//     Drive/Outputs/Out/nCtrl2 <-> Receive PDO 1/Control Word @bit 8
//     Drive/Outputs/Out/nDataOut1 <-> Receive PDO 1/Profile Target Position
//     Enc/Inputs/In/nDataIn1 <-> Transmit PDO 1/Position Actual Value
//     Enc/Inputs/In/nDataIn3 <-> Transmit PDO 1/Touch Probe 1 Positive Value
//     Enc/Inputs/In/nDcInputTime <-> InfoData/DcInputShift
//     Enc/Inputs/In/nState4 @bit 1 <-> WcState/InputToggle
//     Enc/Inputs/In/nState4 <-> WcState/WcState
//     Enc/Inputs/In/nState5 <-> Transmit PDO 1/Touch Probe Status
//     Enc/Inputs/In/nState6 <-> Transmit PDO 1/Touch Probe Status @bit 8
//     Enc/Outputs/Out/nCtrl5 <-> Receive PDO 1/Touch Probe Function
//     Enc/Outputs/Out/nCtrl6 <-> Receive PDO 1/Touch Probe Function @bit 8
//   NC-Task 1 SAF/Axes/Axis180_132 P2M3_SCurlingneedleWhirling <-> Device 3 (EtherCAT)/Box 2 (CU1128)/Term 44 (CU1128-C)/P2M3短卷针旋转[132] (CL3C-EC808AC)
//     Drive/Inputs/In/nDcOutputTime <-> InfoData/DcOutputShift
//     Drive/Inputs/In/nState1 <-> Transmit PDO 1/Status Word
//     Drive/Inputs/In/nState2 <-> Transmit PDO 1/Status Word @bit 8
//     Drive/Inputs/In/nState4 @bit 1 <-> WcState/InputToggle
//     Drive/Inputs/In/nState4 <-> WcState/WcState
//     Drive/Outputs/Out/nCtrl1 <-> Receive PDO 1/Control Word
//     Drive/Outputs/Out/nCtrl2 <-> Receive PDO 1/Control Word @bit 8
//     Drive/Outputs/Out/nDataOut1 <-> Receive PDO 1/Profile Target Position
//     Enc/Inputs/In/nDataIn1 <-> Transmit PDO 1/Position Actual Value
//     Enc/Inputs/In/nDataIn3 <-> Transmit PDO 1/Touch Probe 1 Positive Value
//     Enc/Inputs/In/nDcInputTime <-> InfoData/DcInputShift
//     Enc/Inputs/In/nState4 @bit 1 <-> WcState/InputToggle
//     Enc/Inputs/In/nState4 <-> WcState/WcState
//     Enc/Inputs/In/nState5 <-> Transmit PDO 1/Touch Probe Status
//     Enc/Inputs/In/nState6 <-> Transmit PDO 1/Touch Probe Status @bit 8
//     Enc/Outputs/Out/nCtrl5 <-> Receive PDO 1/Touch Probe Function
//     Enc/Outputs/Out/nCtrl6 <-> Receive PDO 1/Touch Probe Function @bit 8
//   NC-Task 1 SAF/Axes/Axis181_133 P2M3_GluingLine <-> Device 3 (EtherCAT)/Box 2 (CU1128)/Term 44 (CU1128-C)/P2M3侧贴夹平移（ 133）(InoSV660N)
//     Drive/Inputs/In/nDataIn1 <-> Inputs/Following error actual value
//     Drive/Inputs/In/nDcOutputTime <-> InfoData/DcOutputShift
//     Drive/Inputs/In/nState1 <-> Inputs/Statusword
//     Drive/Inputs/In/nState2 <-> Inputs/Statusword @bit 8
//     Drive/Inputs/In/nState4 @bit 1 <-> WcState/InputToggle
//     Drive/Inputs/In/nState4 <-> WcState/WcState
//     Drive/Outputs/Out/nCtrl1 <-> Outputs/Controlword
//     Drive/Outputs/Out/nCtrl2 <-> Outputs/Controlword @bit 8
//     Drive/Outputs/Out/nDataOut1 <-> Outputs/Target position
//     Enc/Inputs/In/nDataIn1 <-> Inputs/Position actual value
//     Enc/Inputs/In/nDataIn3 <-> Inputs/Touch probe pos1 pos value
//     Enc/Inputs/In/nDataIn5 <-> Inputs/Touch probe pos2 pos value
//     Enc/Inputs/In/nDcInputTime <-> InfoData/DcInputShift
//     Enc/Inputs/In/nState4 @bit 1 <-> WcState/InputToggle
//     Enc/Inputs/In/nState4 <-> WcState/WcState
//     Enc/Inputs/In/nState5 <-> Inputs/Touch probe status
//     Enc/Inputs/In/nState6 <-> Inputs/Touch probe status @bit 8
//     Enc/Outputs/Out/nCtrl5 <-> Outputs/Touch probe function
//     Enc/Outputs/Out/nCtrl6 <-> Outputs/Touch probe function @bit 8
//   NC-Task 1 SAF/Axes/Axis182_134 P2M3_GluingWhirling <-> Device 3 (EtherCAT)/Box 2 (CU1128)/Term 44 (CU1128-C)/P2M3侧贴夹旋转[134] (InoSV660N)
//     Drive/Inputs/In/nDataIn1 <-> Inputs/Following error actual value
//     Drive/Inputs/In/nDcOutputTime <-> InfoData/DcOutputShift
//     Drive/Inputs/In/nState1 <-> Inputs/Statusword
//     Drive/Inputs/In/nState2 <-> Inputs/Statusword @bit 8
//     Drive/Inputs/In/nState4 @bit 1 <-> WcState/InputToggle
//     Drive/Inputs/In/nState4 <-> WcState/WcState
//     Drive/Outputs/Out/nCtrl1 <-> Outputs/Controlword
//     Drive/Outputs/Out/nCtrl2 <-> Outputs/Controlword @bit 8
//     Drive/Outputs/Out/nDataOut1 <-> Outputs/Target position
//     Enc/Inputs/In/nDataIn1 <-> Inputs/Position actual value
//     Enc/Inputs/In/nDataIn3 <-> Inputs/Touch probe pos1 pos value
//     Enc/Inputs/In/nDataIn5 <-> Inputs/Touch probe pos2 pos value
//     Enc/Inputs/In/nDcInputTime <-> InfoData/DcInputShift
//     Enc/Inputs/In/nState4 @bit 1 <-> WcState/InputToggle
//     Enc/Inputs/In/nState4 <-> WcState/WcState
//     Enc/Inputs/In/nState5 <-> Inputs/Touch probe status
//     Enc/Inputs/In/nState6 <-> Inputs/Touch probe status @bit 8
//     Enc/Outputs/Out/nCtrl5 <-> Outputs/Touch probe function
//     Enc/Outputs/Out/nCtrl6 <-> Outputs/Touch probe function @bit 8
//   NC-Task 1 SAF/Axes/Axis183_135 P2M3_GluingRetracting <-> Device 3 (EtherCAT)/Box 2 (CU1128)/Term 44 (CU1128-C)/P2M3贴胶头进退[135] (InoSV660N)
//     Drive/Inputs/In/nDataIn1 <-> Inputs/Following error actual value
//     Drive/Inputs/In/nDcOutputTime <-> InfoData/DcOutputShift
//     Drive/Inputs/In/nState1 <-> Inputs/Statusword
//     Drive/Inputs/In/nState2 <-> Inputs/Statusword @bit 8
//     Drive/Inputs/In/nState4 @bit 1 <-> WcState/InputToggle
//     Drive/Inputs/In/nState4 <-> WcState/WcState
//     Drive/Outputs/Out/nCtrl1 <-> Outputs/Controlword
//     Drive/Outputs/Out/nCtrl2 <-> Outputs/Controlword @bit 8
//     Drive/Outputs/Out/nDataOut1 <-> Outputs/Target position
//     Enc/Inputs/In/nDataIn1 <-> Inputs/Position actual value
//     Enc/Inputs/In/nDataIn3 <-> Inputs/Touch probe pos1 pos value
//     Enc/Inputs/In/nDataIn5 <-> Inputs/Touch probe pos2 pos value
//     Enc/Inputs/In/nDcInputTime <-> InfoData/DcInputShift
//     Enc/Inputs/In/nState4 @bit 1 <-> WcState/InputToggle
//     Enc/Inputs/In/nState4 <-> WcState/WcState
//     Enc/Inputs/In/nState5 <-> Inputs/Touch probe status
//     Enc/Inputs/In/nState6 <-> Inputs/Touch probe status @bit 8
//     Enc/Outputs/Out/nCtrl5 <-> Outputs/Touch probe function
//     Enc/Outputs/Out/nCtrl6 <-> Outputs/Touch probe function @bit 8
//   NC-Task 1 SAF/Axes/Axis184_136 P2M3_GluingUpDown <-> Device 3 (EtherCAT)/Box 2 (CU1128)/Term 44 (CU1128-C)/P2M3拉胶升降[136](InoSV660N)
//     Drive/Inputs/In/nDataIn1 <-> Inputs/Following error actual value
//     Drive/Inputs/In/nDcOutputTime <-> InfoData/DcOutputShift
//     Drive/Inputs/In/nState1 <-> Inputs/Statusword
//     Drive/Inputs/In/nState2 <-> Inputs/Statusword @bit 8
//     Drive/Inputs/In/nState4 @bit 1 <-> WcState/InputToggle
//     Drive/Inputs/In/nState4 <-> WcState/WcState
//     Drive/Outputs/Out/nCtrl1 <-> Outputs/Controlword
//     Drive/Outputs/Out/nCtrl2 <-> Outputs/Controlword @bit 8
//     Drive/Outputs/Out/nDataOut1 <-> Outputs/Target position
//     Enc/Inputs/In/nDataIn1 <-> Inputs/Position actual value
//     Enc/Inputs/In/nDataIn3 <-> Inputs/Touch probe pos1 pos value
//     Enc/Inputs/In/nDataIn5 <-> Inputs/Touch probe pos2 pos value
//     Enc/Inputs/In/nDcInputTime <-> InfoData/DcInputShift
//     Enc/Inputs/In/nState4 @bit 1 <-> WcState/InputToggle
//     Enc/Inputs/In/nState4 <-> WcState/WcState
//     Enc/Inputs/In/nState5 <-> Inputs/Touch probe status
//     Enc/Inputs/In/nState6 <-> Inputs/Touch probe status @bit 8
//     Enc/Outputs/Out/nCtrl5 <-> Outputs/Touch probe function
//     Enc/Outputs/Out/nCtrl6 <-> Outputs/Touch probe function @bit 8
//   NC-Task 1 SAF/Axes/Axis187_160 P3M1_ColdpreLine <-> Device 3 (EtherCAT)/P2M1冷压上料夹平移 [160（热压）](InoSV660N)
//     Drive/Inputs/In/nDataIn1 <-> Inputs/Following error actual value
//     Drive/Inputs/In/nDcOutputTime <-> InfoData/DcOutputShift
//     Drive/Inputs/In/nState1 <-> Inputs/Statusword
//     Drive/Inputs/In/nState2 <-> Inputs/Statusword @bit 8
//     Drive/Inputs/In/nState4 @bit 1 <-> WcState/InputToggle
//     Drive/Inputs/In/nState4 <-> WcState/WcState
//     Drive/Outputs/Out/nCtrl1 <-> Outputs/Controlword
//     Drive/Outputs/Out/nCtrl2 <-> Outputs/Controlword @bit 8
//     Drive/Outputs/Out/nDataOut1 <-> Outputs/Target position
//     Enc/Inputs/In/nDataIn1 <-> Inputs/Position actual value
//     Enc/Inputs/In/nDataIn3 <-> Inputs/Touch probe pos1 pos value
//     Enc/Inputs/In/nDataIn5 <-> Inputs/Touch probe pos2 pos value
//     Enc/Inputs/In/nDcInputTime <-> InfoData/DcInputShift
//     Enc/Inputs/In/nState4 @bit 1 <-> WcState/InputToggle
//     Enc/Inputs/In/nState4 <-> WcState/WcState
//     Enc/Inputs/In/nState5 <-> Inputs/Touch probe status
//     Enc/Inputs/In/nState6 <-> Inputs/Touch probe status @bit 8
//     Enc/Outputs/Out/nCtrl5 <-> Outputs/Touch probe function
//     Enc/Outputs/Out/nCtrl6 <-> Outputs/Touch probe function @bit 8
//   NC-Task 1 SAF/Axes/Axis188_161 P3M1_ColdpreRetracting <-> Device 3 (EtherCAT)/Box 2 (CU1128)/Term 44 (CU1128-C)/P2M2冷压上料夹进退[161（热压）] (InoSV660N)
//     Drive/Inputs/In/nDataIn1 <-> Inputs/Following error actual value
//     Drive/Inputs/In/nDcOutputTime <-> InfoData/DcOutputShift
//     Drive/Inputs/In/nState1 <-> Inputs/Statusword
//     Drive/Inputs/In/nState2 <-> Inputs/Statusword @bit 8
//     Drive/Inputs/In/nState4 @bit 1 <-> WcState/InputToggle
//     Drive/Inputs/In/nState4 <-> WcState/WcState
//     Drive/Outputs/Out/nCtrl1 <-> Outputs/Controlword
//     Drive/Outputs/Out/nCtrl2 <-> Outputs/Controlword @bit 8
//     Drive/Outputs/Out/nDataOut1 <-> Outputs/Target position
//     Enc/Inputs/In/nDataIn1 <-> Inputs/Position actual value
//     Enc/Inputs/In/nDataIn3 <-> Inputs/Touch probe pos1 pos value
//     Enc/Inputs/In/nDataIn5 <-> Inputs/Touch probe pos2 pos value
//     Enc/Inputs/In/nDcInputTime <-> InfoData/DcInputShift
//     Enc/Inputs/In/nState4 @bit 1 <-> WcState/InputToggle
//     Enc/Inputs/In/nState4 <-> WcState/WcState
//     Enc/Inputs/In/nState5 <-> Inputs/Touch probe status
//     Enc/Inputs/In/nState6 <-> Inputs/Touch probe status @bit 8
//     Enc/Outputs/Out/nCtrl5 <-> Outputs/Touch probe function
//     Enc/Outputs/Out/nCtrl6 <-> Outputs/Touch probe function @bit 8
//   NC-Task 1 SAF/Axes/Axis189_162 P3M1_ColdpreWhirling <-> Device 3 (EtherCAT)/Box 2 (CU1128)/Term 44 (CU1128-C)/P2M2冷压上料夹旋转[162（热压）] (InoSV660N)
//     Drive/Inputs/In/nDataIn1 <-> Inputs/Following error actual value
//     Drive/Inputs/In/nDcOutputTime <-> InfoData/DcOutputShift
//     Drive/Inputs/In/nState1 <-> Inputs/Statusword
//     Drive/Inputs/In/nState2 <-> Inputs/Statusword @bit 8
//     Drive/Inputs/In/nState4 @bit 1 <-> WcState/InputToggle
//     Drive/Inputs/In/nState4 <-> WcState/WcState
//     Drive/Outputs/Out/nCtrl1 <-> Outputs/Controlword
//     Drive/Outputs/Out/nCtrl2 <-> Outputs/Controlword @bit 8
//     Drive/Outputs/Out/nDataOut1 <-> Outputs/Target position
//     Enc/Inputs/In/nDataIn1 <-> Inputs/Position actual value
//     Enc/Inputs/In/nDataIn3 <-> Inputs/Touch probe pos1 pos value
//     Enc/Inputs/In/nDataIn5 <-> Inputs/Touch probe pos2 pos value
//     Enc/Inputs/In/nDcInputTime <-> InfoData/DcInputShift
//     Enc/Inputs/In/nState4 @bit 1 <-> WcState/InputToggle
//     Enc/Inputs/In/nState4 <-> WcState/WcState
//     Enc/Inputs/In/nState5 <-> Inputs/Touch probe status
//     Enc/Inputs/In/nState6 <-> Inputs/Touch probe status @bit 8
//     Enc/Outputs/Out/nCtrl5 <-> Outputs/Touch probe function
//     Enc/Outputs/Out/nCtrl6 <-> Outputs/Touch probe function @bit 8
//   NC-Task 1 SAF/Axes/Axis190_163 P3M1_ColdpreUpDown <-> Device 3 (EtherCAT)/Box 2 (CU1128)/Term 44 (CU1128-C)/P2M2冷压上料夹升降[163（热压）] (InoSV660N)
//     Drive/Inputs/In/nDataIn1 <-> Inputs/Following error actual value
//     Drive/Inputs/In/nDcOutputTime <-> InfoData/DcOutputShift
//     Drive/Inputs/In/nState1 <-> Inputs/Statusword
//     Drive/Inputs/In/nState2 <-> Inputs/Statusword @bit 8
//     Drive/Inputs/In/nState4 @bit 1 <-> WcState/InputToggle
//     Drive/Inputs/In/nState4 <-> WcState/WcState
//     Drive/Outputs/Out/nCtrl1 <-> Outputs/Controlword
//     Drive/Outputs/Out/nCtrl2 <-> Outputs/Controlword @bit 8
//     Drive/Outputs/Out/nDataOut1 <-> Outputs/Target position
//     Enc/Inputs/In/nDataIn1 <-> Inputs/Position actual value
//     Enc/Inputs/In/nDataIn3 <-> Inputs/Touch probe pos1 pos value
//     Enc/Inputs/In/nDataIn5 <-> Inputs/Touch probe pos2 pos value
//     Enc/Inputs/In/nDcInputTime <-> InfoData/DcInputShift
//     Enc/Inputs/In/nState4 @bit 1 <-> WcState/InputToggle
//     Enc/Inputs/In/nState4 <-> WcState/WcState
//     Enc/Inputs/In/nState5 <-> Inputs/Touch probe status
//     Enc/Inputs/In/nState6 <-> Inputs/Touch probe status @bit 8
//     Enc/Outputs/Out/nCtrl5 <-> Outputs/Touch probe function
//     Enc/Outputs/Out/nCtrl6 <-> Outputs/Touch probe function @bit 8
//   NC-Task 1 SAF/Axes/Axis191_164 P3M1_ColdpreSupPlateLine <-> Device 3 (EtherCAT)/Box 2 (CU1128)/Term 24 (CU1128-B)/冷压托板开合[164] (CL3C-EC503)
//     Drive/Inputs/In/nDcOutputTime <-> InfoData/DcOutputShift
//     Drive/Inputs/In/nState1 <-> Transmit PDO 1/Status Word
//     Drive/Inputs/In/nState2 <-> Transmit PDO 1/Status Word @bit 8
//     Drive/Inputs/In/nState4 @bit 1 <-> WcState/InputToggle
//     Drive/Inputs/In/nState4 <-> WcState/WcState
//     Drive/Outputs/Out/nCtrl1 <-> Receive PDO 1/Control Word
//     Drive/Outputs/Out/nCtrl2 <-> Receive PDO 1/Control Word @bit 8
//     Drive/Outputs/Out/nDataOut1 <-> Receive PDO 1/Profile Target Position
//     Enc/Inputs/In/nDataIn1 <-> Transmit PDO 1/Position Actual Value
//     Enc/Inputs/In/nDataIn3 <-> Transmit PDO 1/Touch Probe 1 Positive Value
//     Enc/Inputs/In/nDcInputTime <-> InfoData/DcInputShift
//     Enc/Inputs/In/nState4 @bit 1 <-> WcState/InputToggle
//     Enc/Inputs/In/nState4 <-> WcState/WcState
//     Enc/Inputs/In/nState5 <-> Transmit PDO 1/Touch Probe Status
//     Enc/Inputs/In/nState6 <-> Transmit PDO 1/Touch Probe Status @bit 8
//     Enc/Outputs/Out/nCtrl5 <-> Receive PDO 1/Touch Probe Function
//     Enc/Outputs/Out/nCtrl6 <-> Receive PDO 1/Touch Probe Function @bit 8
//   NC-Task 1 SAF/Axes/Axis192_165 P3M1_ColdpreActuated <-> Device 3 (EtherCAT)/Box 2 (CU1128)/Term 24 (CU1128-B)/冷压驱动[165](InoSV660N)
//     Drive/Inputs/In/nDataIn1 <-> Inputs/Following error actual value
//     Drive/Inputs/In/nDcOutputTime <-> InfoData/DcOutputShift
//     Drive/Inputs/In/nState1 <-> Inputs/Statusword
//     Drive/Inputs/In/nState2 <-> Inputs/Statusword @bit 8
//     Drive/Inputs/In/nState4 @bit 1 <-> WcState/InputToggle
//     Drive/Inputs/In/nState4 <-> WcState/WcState
//     Drive/Outputs/Out/nCtrl1 <-> Outputs/Controlword
//     Drive/Outputs/Out/nCtrl2 <-> Outputs/Controlword @bit 8
//     Drive/Outputs/Out/nDataOut1 <-> Outputs/Target position
//     Enc/Inputs/In/nDataIn1 <-> Inputs/Position actual value
//     Enc/Inputs/In/nDataIn3 <-> Inputs/Touch probe pos1 pos value
//     Enc/Inputs/In/nDataIn5 <-> Inputs/Touch probe pos2 pos value
//     Enc/Inputs/In/nDcInputTime <-> InfoData/DcInputShift
//     Enc/Inputs/In/nState4 @bit 1 <-> WcState/InputToggle
//     Enc/Inputs/In/nState4 <-> WcState/WcState
//     Enc/Inputs/In/nState5 <-> Inputs/Touch probe status
//     Enc/Inputs/In/nState6 <-> Inputs/Touch probe status @bit 8
//     Enc/Outputs/Out/nCtrl5 <-> Outputs/Touch probe function
//     Enc/Outputs/Out/nCtrl6 <-> Outputs/Touch probe function @bit 8
//   NC-Task 1 SAF/Axes/Axis193_166 P3_M2_OvenCarrying <-> Device 3 (EtherCAT)/Box 2 (CU1128)/Term 24 (CU1128-B)/烤箱上料夹搬运[166] (InoSV660N)
//     Drive/Inputs/In/nDataIn1 <-> Inputs/Following error actual value
//     Drive/Inputs/In/nDcOutputTime <-> InfoData/DcOutputShift
//     Drive/Inputs/In/nState1 <-> Inputs/Statusword
//     Drive/Inputs/In/nState2 <-> Inputs/Statusword @bit 8
//     Drive/Inputs/In/nState4 @bit 1 <-> WcState/InputToggle
//     Drive/Inputs/In/nState4 <-> WcState/WcState
//     Drive/Outputs/Out/nCtrl1 <-> Outputs/Controlword
//     Drive/Outputs/Out/nCtrl2 <-> Outputs/Controlword @bit 8
//     Drive/Outputs/Out/nDataOut1 <-> Outputs/Target position
//     Enc/Inputs/In/nDataIn1 <-> Inputs/Position actual value
//     Enc/Inputs/In/nDataIn3 <-> Inputs/Touch probe pos1 pos value
//     Enc/Inputs/In/nDataIn5 <-> Inputs/Touch probe pos2 pos value
//     Enc/Inputs/In/nDcInputTime <-> InfoData/DcInputShift
//     Enc/Inputs/In/nState4 @bit 1 <-> WcState/InputToggle
//     Enc/Inputs/In/nState4 <-> WcState/WcState
//     Enc/Inputs/In/nState5 <-> Inputs/Touch probe status
//     Enc/Inputs/In/nState6 <-> Inputs/Touch probe status @bit 8
//     Enc/Outputs/Out/nCtrl5 <-> Outputs/Touch probe function
//     Enc/Outputs/Out/nCtrl6 <-> Outputs/Touch probe function @bit 8
//   NC-Task 1 SAF/Axes/Axis194_167 P3_M2_OvenRetracting <-> Device 3 (EtherCAT)/Box 2 (CU1128)/Term 24 (CU1128-B)/烤箱上料夹进退[167] (InoSV660N)
//     Drive/Inputs/In/nDataIn1 <-> Inputs/Following error actual value
//     Drive/Inputs/In/nDcOutputTime <-> InfoData/DcOutputShift
//     Drive/Inputs/In/nState1 <-> Inputs/Statusword
//     Drive/Inputs/In/nState2 <-> Inputs/Statusword @bit 8
//     Drive/Inputs/In/nState4 @bit 1 <-> WcState/InputToggle
//     Drive/Inputs/In/nState4 <-> WcState/WcState
//     Drive/Outputs/Out/nCtrl1 <-> Outputs/Controlword
//     Drive/Outputs/Out/nCtrl2 <-> Outputs/Controlword @bit 8
//     Drive/Outputs/Out/nDataOut1 <-> Outputs/Target position
//     Enc/Inputs/In/nDataIn1 <-> Inputs/Position actual value
//     Enc/Inputs/In/nDataIn3 <-> Inputs/Touch probe pos1 pos value
//     Enc/Inputs/In/nDataIn5 <-> Inputs/Touch probe pos2 pos value
//     Enc/Inputs/In/nDcInputTime <-> InfoData/DcInputShift
//     Enc/Inputs/In/nState4 @bit 1 <-> WcState/InputToggle
//     Enc/Inputs/In/nState4 <-> WcState/WcState
//     Enc/Inputs/In/nState5 <-> Inputs/Touch probe status
//     Enc/Inputs/In/nState6 <-> Inputs/Touch probe status @bit 8
//     Enc/Outputs/Out/nCtrl5 <-> Outputs/Touch probe function
//     Enc/Outputs/Out/nCtrl6 <-> Outputs/Touch probe function @bit 8
//   NC-Task 1 SAF/Axes/Axis195_168 P3_M2_OvenUpDown <-> Device 3 (EtherCAT)/Box 2 (CU1128)/Term 24 (CU1128-B)/烤箱上料夹升降[168](InoSV660N)
//     Drive/Inputs/In/nDataIn1 <-> Inputs/Following error actual value
//     Drive/Inputs/In/nDcOutputTime <-> InfoData/DcOutputShift
//     Drive/Inputs/In/nState1 <-> Inputs/Statusword
//     Drive/Inputs/In/nState2 <-> Inputs/Statusword @bit 8
//     Drive/Inputs/In/nState4 @bit 1 <-> WcState/InputToggle
//     Drive/Inputs/In/nState4 <-> WcState/WcState
//     Drive/Outputs/Out/nCtrl1 <-> Outputs/Controlword
//     Drive/Outputs/Out/nCtrl2 <-> Outputs/Controlword @bit 8
//     Drive/Outputs/Out/nDataOut1 <-> Outputs/Target position
//     Enc/Inputs/In/nDataIn1 <-> Inputs/Position actual value
//     Enc/Inputs/In/nDataIn3 <-> Inputs/Touch probe pos1 pos value
//     Enc/Inputs/In/nDataIn5 <-> Inputs/Touch probe pos2 pos value
//     Enc/Inputs/In/nDcInputTime <-> InfoData/DcInputShift
//     Enc/Inputs/In/nState4 @bit 1 <-> WcState/InputToggle
//     Enc/Inputs/In/nState4 <-> WcState/WcState
//     Enc/Inputs/In/nState5 <-> Inputs/Touch probe status
//     Enc/Inputs/In/nState6 <-> Inputs/Touch probe status @bit 8
//     Enc/Outputs/Out/nCtrl5 <-> Outputs/Touch probe function
//     Enc/Outputs/Out/nCtrl6 <-> Outputs/Touch probe function @bit 8
//   NC-Task 1 SAF/Axes/Axis196_169 P3_M3_HotPressingLine <-> Device 3 (EtherCAT)/Box 2 (CU1128)/Term 24 (CU1128-B)/热压托板开合[169] (CL3C-EC503)
//     Drive/Inputs/In/nDcOutputTime <-> InfoData/DcOutputShift
//     Drive/Inputs/In/nState1 <-> Transmit PDO 1/Status Word
//     Drive/Inputs/In/nState2 <-> Transmit PDO 1/Status Word @bit 8
//     Drive/Inputs/In/nState4 @bit 1 <-> WcState/InputToggle
//     Drive/Inputs/In/nState4 <-> WcState/WcState
//     Drive/Outputs/Out/nCtrl1 <-> Receive PDO 1/Control Word
//     Drive/Outputs/Out/nCtrl2 <-> Receive PDO 1/Control Word @bit 8
//     Drive/Outputs/Out/nDataOut1 <-> Receive PDO 1/Profile Target Position
//     Enc/Inputs/In/nDataIn1 <-> Transmit PDO 1/Position Actual Value
//     Enc/Inputs/In/nDataIn3 <-> Transmit PDO 1/Touch Probe 1 Positive Value
//     Enc/Inputs/In/nDcInputTime <-> InfoData/DcInputShift
//     Enc/Inputs/In/nState4 @bit 1 <-> WcState/InputToggle
//     Enc/Inputs/In/nState4 <-> WcState/WcState
//     Enc/Inputs/In/nState5 <-> Transmit PDO 1/Touch Probe Status
//     Enc/Inputs/In/nState6 <-> Transmit PDO 1/Touch Probe Status @bit 8
//     Enc/Outputs/Out/nCtrl5 <-> Receive PDO 1/Touch Probe Function
//     Enc/Outputs/Out/nCtrl6 <-> Receive PDO 1/Touch Probe Function @bit 8
//   NC-Task 1 SAF/Axes/Axis197_170 P3_M3_HotPressingActuated <-> Device 3 (EtherCAT)/Box 2 (CU1128)/Term 24 (CU1128-B)/热压驱动[170] (InoSV660N)
//     Drive/Inputs/In/nDataIn1 <-> Inputs/Following error actual value
//     Drive/Inputs/In/nDcOutputTime <-> InfoData/DcOutputShift
//     Drive/Inputs/In/nState1 <-> Inputs/Statusword
//     Drive/Inputs/In/nState2 <-> Inputs/Statusword @bit 8
//     Drive/Inputs/In/nState4 @bit 1 <-> WcState/InputToggle
//     Drive/Inputs/In/nState4 <-> WcState/WcState
//     Drive/Outputs/Out/nCtrl1 <-> Outputs/Controlword
//     Drive/Outputs/Out/nCtrl2 <-> Outputs/Controlword @bit 8
//     Drive/Outputs/Out/nDataOut1 <-> Outputs/Target position
//     Enc/Inputs/In/nDataIn1 <-> Inputs/Position actual value
//     Enc/Inputs/In/nDataIn3 <-> Inputs/Touch probe pos1 pos value
//     Enc/Inputs/In/nDataIn5 <-> Inputs/Touch probe pos2 pos value
//     Enc/Inputs/In/nDcInputTime <-> InfoData/DcInputShift
//     Enc/Inputs/In/nState4 @bit 1 <-> WcState/InputToggle
//     Enc/Inputs/In/nState4 <-> WcState/WcState
//     Enc/Inputs/In/nState5 <-> Inputs/Touch probe status
//     Enc/Inputs/In/nState6 <-> Inputs/Touch probe status @bit 8
//     Enc/Outputs/Out/nCtrl5 <-> Outputs/Touch probe function
//     Enc/Outputs/Out/nCtrl6 <-> Outputs/Touch probe function @bit 8
//   NC-Task 1 SAF/Axes/Axis198_171  P3_M4_WeighLine <-> Device 3 (EtherCAT)/Box 2 (CU1128)/Term 24 (CU1128-B)/称重上料夹平移[171] (InoSV660N)
//     Drive/Inputs/In/nDataIn1 <-> Inputs/Following error actual value
//     Drive/Inputs/In/nDcOutputTime <-> InfoData/DcOutputShift
//     Drive/Inputs/In/nState1 <-> Inputs/Statusword
//     Drive/Inputs/In/nState2 <-> Inputs/Statusword @bit 8
//     Drive/Inputs/In/nState4 @bit 1 <-> WcState/InputToggle
//     Drive/Inputs/In/nState4 <-> WcState/WcState
//     Drive/Outputs/Out/nCtrl1 <-> Outputs/Controlword
//     Drive/Outputs/Out/nCtrl2 <-> Outputs/Controlword @bit 8
//     Drive/Outputs/Out/nDataOut1 <-> Outputs/Target position
//     Enc/Inputs/In/nDataIn1 <-> Inputs/Position actual value
//     Enc/Inputs/In/nDataIn3 <-> Inputs/Touch probe pos1 pos value
//     Enc/Inputs/In/nDataIn5 <-> Inputs/Touch probe pos2 pos value
//     Enc/Inputs/In/nDcInputTime <-> InfoData/DcInputShift
//     Enc/Inputs/In/nState4 @bit 1 <-> WcState/InputToggle
//     Enc/Inputs/In/nState4 <-> WcState/WcState
//     Enc/Inputs/In/nState5 <-> Inputs/Touch probe status
//     Enc/Inputs/In/nState6 <-> Inputs/Touch probe status @bit 8
//     Enc/Outputs/Out/nCtrl5 <-> Outputs/Touch probe function
//     Enc/Outputs/Out/nCtrl6 <-> Outputs/Touch probe function @bit 8
//   NC-Task 1 SAF/Axes/Axis199_172 P3_M4_WeighUpDown <-> Device 3 (EtherCAT)/Box 2 (CU1128)/Term 24 (CU1128-B)/称重上料夹升降[172](InoSV660N)
//     Drive/Inputs/In/nDataIn1 <-> Inputs/Following error actual value
//     Drive/Inputs/In/nDcOutputTime <-> InfoData/DcOutputShift
//     Drive/Inputs/In/nState1 <-> Inputs/Statusword
//     Drive/Inputs/In/nState2 <-> Inputs/Statusword @bit 8
//     Drive/Inputs/In/nState4 @bit 1 <-> WcState/InputToggle
//     Drive/Inputs/In/nState4 <-> WcState/WcState
//     Drive/Outputs/Out/nCtrl1 <-> Outputs/Controlword
//     Drive/Outputs/Out/nCtrl2 <-> Outputs/Controlword @bit 8
//     Drive/Outputs/Out/nDataOut1 <-> Outputs/Target position
//     Enc/Inputs/In/nDataIn1 <-> Inputs/Position actual value
//     Enc/Inputs/In/nDataIn3 <-> Inputs/Touch probe pos1 pos value
//     Enc/Inputs/In/nDataIn5 <-> Inputs/Touch probe pos2 pos value
//     Enc/Inputs/In/nDcInputTime <-> InfoData/DcInputShift
//     Enc/Inputs/In/nState4 @bit 1 <-> WcState/InputToggle
//     Enc/Inputs/In/nState4 <-> WcState/WcState
//     Enc/Inputs/In/nState5 <-> Inputs/Touch probe status
//     Enc/Inputs/In/nState6 <-> Inputs/Touch probe status @bit 8
//     Enc/Outputs/Out/nCtrl5 <-> Outputs/Touch probe function
//     Enc/Outputs/Out/nCtrl6 <-> Outputs/Touch probe function @bit 8
//   NC-Task 1 SAF/Axes/Axis200_173 P3_M4_WeighWhirling <-> Device 3 (EtherCAT)/Box 2 (CU1128)/Term 24 (CU1128-B)/称重上料夹旋转[173] (InoSV660N)
//     Drive/Inputs/In/nDataIn1 <-> Inputs/Following error actual value
//     Drive/Inputs/In/nDcOutputTime <-> InfoData/DcOutputShift
//     Drive/Inputs/In/nState1 <-> Inputs/Statusword
//     Drive/Inputs/In/nState2 <-> Inputs/Statusword @bit 8
//     Drive/Inputs/In/nState4 @bit 1 <-> WcState/InputToggle
//     Drive/Inputs/In/nState4 <-> WcState/WcState
//     Drive/Outputs/Out/nCtrl1 <-> Outputs/Controlword
//     Drive/Outputs/Out/nCtrl2 <-> Outputs/Controlword @bit 8
//     Drive/Outputs/Out/nDataOut1 <-> Outputs/Target position
//     Enc/Inputs/In/nDataIn1 <-> Inputs/Position actual value
//     Enc/Inputs/In/nDataIn3 <-> Inputs/Touch probe pos1 pos value
//     Enc/Inputs/In/nDataIn5 <-> Inputs/Touch probe pos2 pos value
//     Enc/Inputs/In/nDcInputTime <-> InfoData/DcInputShift
//     Enc/Inputs/In/nState4 @bit 1 <-> WcState/InputToggle
//     Enc/Inputs/In/nState4 <-> WcState/WcState
//     Enc/Inputs/In/nState5 <-> Inputs/Touch probe status
//     Enc/Inputs/In/nState6 <-> Inputs/Touch probe status @bit 8
//     Enc/Outputs/Out/nCtrl5 <-> Outputs/Touch probe function
//     Enc/Outputs/Out/nCtrl6 <-> Outputs/Touch probe function @bit 8
//   NC-Task 1 SAF/Axes/Axis201_174 P3_M4_SortingoutCarrying <-> Device 3 (EtherCAT)/Box 2 (CU1128)/Term 24 (CU1128-B)/电芯分选夹搬运[174](InoSV660N)
//     Drive/Inputs/In/nDataIn1 <-> Inputs/Following error actual value
//     Drive/Inputs/In/nDcOutputTime <-> InfoData/DcOutputShift
//     Drive/Inputs/In/nState1 <-> Inputs/Statusword
//     Drive/Inputs/In/nState2 <-> Inputs/Statusword @bit 8
//     Drive/Inputs/In/nState4 @bit 1 <-> WcState/InputToggle
//     Drive/Inputs/In/nState4 <-> WcState/WcState
//     Drive/Outputs/Out/nCtrl1 <-> Outputs/Controlword
//     Drive/Outputs/Out/nCtrl2 <-> Outputs/Controlword @bit 8
//     Drive/Outputs/Out/nDataOut1 <-> Outputs/Target position
//     Enc/Inputs/In/nDataIn1 <-> Inputs/Position actual value
//     Enc/Inputs/In/nDataIn3 <-> Inputs/Touch probe pos1 pos value
//     Enc/Inputs/In/nDataIn5 <-> Inputs/Touch probe pos2 pos value
//     Enc/Inputs/In/nDcInputTime <-> InfoData/DcInputShift
//     Enc/Inputs/In/nState4 @bit 1 <-> WcState/InputToggle
//     Enc/Inputs/In/nState4 <-> WcState/WcState
//     Enc/Inputs/In/nState5 <-> Inputs/Touch probe status
//     Enc/Inputs/In/nState6 <-> Inputs/Touch probe status @bit 8
//     Enc/Outputs/Out/nCtrl5 <-> Outputs/Touch probe function
//     Enc/Outputs/Out/nCtrl6 <-> Outputs/Touch probe function @bit 8
//   NC-Task 1 SAF/Axes/Axis202_175 P3_M4_SortingoutUpDown <-> Device 3 (EtherCAT)/Box 2 (CU1128)/Term 24 (CU1128-B)/电芯分选夹升降[175] (InoSV660N)
//     Drive/Inputs/In/nDataIn1 <-> Inputs/Following error actual value
//     Drive/Inputs/In/nDcOutputTime <-> InfoData/DcOutputShift
//     Drive/Inputs/In/nState1 <-> Inputs/Statusword
//     Drive/Inputs/In/nState2 <-> Inputs/Statusword
//     Drive/Inputs/In/nState4 @bit 1 <-> WcState/InputToggle
//     Drive/Inputs/In/nState4 <-> WcState/WcState
//     Drive/Outputs/Out/nCtrl1 <-> Outputs/Controlword
//     Drive/Outputs/Out/nCtrl2 <-> Outputs/Controlword @bit 8
//     Drive/Outputs/Out/nDataOut1 <-> Outputs/Target position
//     Enc/Inputs/In/nDataIn1 <-> Inputs/Position actual value
//     Enc/Inputs/In/nDataIn3 <-> Inputs/Touch probe pos1 pos value
//     Enc/Inputs/In/nDataIn5 <-> Inputs/Touch probe pos2 pos value
//     Enc/Inputs/In/nDcInputTime <-> InfoData/DcInputShift
//     Enc/Inputs/In/nState4 @bit 1 <-> WcState/InputToggle
//     Enc/Inputs/In/nState4 <-> WcState/WcState
//     Enc/Inputs/In/nState5 <-> Inputs/Touch probe status
//     Enc/Inputs/In/nState6 <-> Inputs/Touch probe status @bit 8
//     Enc/Outputs/Out/nCtrl5 <-> Outputs/Touch probe function
//     Enc/Outputs/Out/nCtrl6 <-> Outputs/Touch probe function @bit 8
//   NC-Task 1 SAF/Axes/Axis203_176 P3_M4_OffloadingCarrying <-> Device 3 (EtherCAT)/Box 2 (CU1128)/Term 24 (CU1128-B)/电芯下料夹搬运[176] (InoSV660N)
//     Drive/Inputs/In/nDataIn1 <-> Inputs/Following error actual value
//     Drive/Inputs/In/nDcOutputTime <-> InfoData/DcOutputShift
//     Drive/Inputs/In/nState1 <-> Inputs/Statusword
//     Drive/Inputs/In/nState2 <-> Inputs/Statusword @bit 8
//     Drive/Inputs/In/nState4 @bit 1 <-> WcState/InputToggle
//     Drive/Inputs/In/nState4 <-> WcState/WcState
//     Drive/Outputs/Out/nCtrl1 <-> Outputs/Controlword
//     Drive/Outputs/Out/nCtrl2 <-> Outputs/Controlword @bit 8
//     Drive/Outputs/Out/nDataOut1 <-> Outputs/Target position
//     Enc/Inputs/In/nDataIn1 <-> Inputs/Position actual value
//     Enc/Inputs/In/nDataIn3 <-> Inputs/Touch probe pos1 pos value
//     Enc/Inputs/In/nDataIn5 <-> Inputs/Touch probe pos2 pos value
//     Enc/Inputs/In/nDcInputTime <-> InfoData/DcInputShift
//     Enc/Inputs/In/nState4 @bit 1 <-> WcState/InputToggle
//     Enc/Inputs/In/nState4 <-> WcState/WcState
//     Enc/Inputs/In/nState5 <-> Inputs/Touch probe status
//     Enc/Inputs/In/nState6 <-> Inputs/Touch probe status @bit 8
//     Enc/Outputs/Out/nCtrl5 <-> Outputs/Touch probe function
//     Enc/Outputs/Out/nCtrl6 <-> Outputs/Touch probe function @bit 8
//   NC-Task 1 SAF/Axes/Axis204_177 P3_M4_OffloadingUpDown <-> Device 3 (EtherCAT)/Box 2 (CU1128)/Term 24 (CU1128-B)/电芯下料夹升降[177] (InoSV660N)
//     Drive/Inputs/In/nDataIn1 <-> Inputs/Following error actual value
//     Drive/Inputs/In/nDcOutputTime <-> InfoData/DcOutputShift
//     Drive/Inputs/In/nState1 <-> Inputs/Statusword
//     Drive/Inputs/In/nState2 <-> Inputs/Statusword @bit 8
//     Drive/Inputs/In/nState4 @bit 1 <-> WcState/InputToggle
//     Drive/Inputs/In/nState4 <-> WcState/WcState
//     Drive/Outputs/Out/nCtrl1 <-> Outputs/Controlword
//     Drive/Outputs/Out/nCtrl2 <-> Outputs/Controlword @bit 8
//     Drive/Outputs/Out/nDataOut1 <-> Outputs/Target position
//     Enc/Inputs/In/nDataIn1 <-> Inputs/Position actual value
//     Enc/Inputs/In/nDataIn3 <-> Inputs/Touch probe pos1 pos value
//     Enc/Inputs/In/nDataIn5 <-> Inputs/Touch probe pos2 pos value
//     Enc/Inputs/In/nDcInputTime <-> InfoData/DcInputShift
//     Enc/Inputs/In/nState4 @bit 1 <-> WcState/InputToggle
//     Enc/Inputs/In/nState4 <-> WcState/WcState
//     Enc/Inputs/In/nState5 <-> Inputs/Touch probe status
//     Enc/Inputs/In/nState6 <-> Inputs/Touch probe status @bit 8
//     Enc/Outputs/Out/nCtrl5 <-> Outputs/Touch probe function
//     Enc/Outputs/Out/nCtrl6 <-> Outputs/Touch probe function @bit 8
//   NC-Task 1 SAF/Axes/Axis205_178 P3_TapeAdvance <-> Device 3 (EtherCAT)/Box 2 (CU1128)/Term 24 (CU1128-B)/贴胶头进退 [178](InoSV660N)
//     Drive/Inputs/In/nDataIn1 <-> Inputs/Following error actual value
//     Drive/Inputs/In/nDataIn3[0] <-> Inputs/Torque actual value
//     Drive/Inputs/In/nDcOutputTime <-> InfoData/DcOutputShift
//     Drive/Inputs/In/nState1 <-> Inputs/Statusword
//     Drive/Inputs/In/nState2 <-> Inputs/Statusword @bit 8
//     Drive/Inputs/In/nState4 @bit 1 <-> WcState/InputToggle
//     Drive/Inputs/In/nState4 <-> WcState/WcState
//     Drive/Outputs/Out/nCtrl1 <-> Outputs/Controlword
//     Drive/Outputs/Out/nCtrl2 <-> Outputs/Controlword @bit 8
//     Drive/Outputs/Out/nDataOut1 <-> Outputs/Target position
//     Enc/Inputs/In/nDataIn1 <-> Inputs/Position actual value
//     Enc/Inputs/In/nDataIn3 <-> Inputs/Touch probe pos1 pos value
//     Enc/Inputs/In/nDataIn5 <-> Inputs/Touch probe pos2 pos value
//     Enc/Inputs/In/nDcInputTime <-> InfoData/DcInputShift
//     Enc/Inputs/In/nState4 @bit 1 <-> WcState/InputToggle
//     Enc/Inputs/In/nState4 <-> WcState/WcState
//     Enc/Inputs/In/nState5 <-> Inputs/Touch probe status
//     Enc/Inputs/In/nState6 <-> Inputs/Touch probe status @bit 8
//     Enc/Outputs/Out/nCtrl5 <-> Outputs/Touch probe function
//     Enc/Outputs/Out/nCtrl6 <-> Outputs/Touch probe function @bit 8
//   NC-Task 1 SAF/Axes/Axis206_179 P3_TapeTranslation <-> Device 3 (EtherCAT)/Box 2 (CU1128)/Term 24 (CU1128-B)/贴胶平移[179](InoSV660N)
//     Drive/Inputs/In/nDataIn1 <-> Inputs/Following error actual value
//     Drive/Inputs/In/nDataIn3[0] <-> Inputs/Torque actual value
//     Drive/Inputs/In/nDcOutputTime <-> InfoData/DcOutputShift
//     Drive/Inputs/In/nState1 <-> Inputs/Statusword
//     Drive/Inputs/In/nState2 <-> Inputs/Statusword @bit 8
//     Drive/Inputs/In/nState4 @bit 1 <-> WcState/InputToggle
//     Drive/Inputs/In/nState4 <-> WcState/WcState
//     Drive/Outputs/Out/nCtrl1 <-> Outputs/Controlword
//     Drive/Outputs/Out/nCtrl2 <-> Outputs/Controlword @bit 8
//     Drive/Outputs/Out/nDataOut1 <-> Outputs/Target position
//     Enc/Inputs/In/nDataIn1 <-> Inputs/Position actual value
//     Enc/Inputs/In/nDataIn3 <-> Inputs/Touch probe pos1 pos value
//     Enc/Inputs/In/nDataIn5 <-> Inputs/Touch probe pos2 pos value
//     Enc/Inputs/In/nDcInputTime <-> InfoData/DcInputShift
//     Enc/Inputs/In/nState4 @bit 1 <-> WcState/InputToggle
//     Enc/Inputs/In/nState4 <-> WcState/WcState
//     Enc/Inputs/In/nState5 <-> Inputs/Touch probe status
//     Enc/Inputs/In/nState6 <-> Inputs/Touch probe status @bit 8
//     Enc/Outputs/Out/nCtrl5 <-> Outputs/Touch probe function
//     Enc/Outputs/Out/nCtrl6 <-> Outputs/Touch probe function @bit 8
//   NC-Task 1 SAF/Axes/Axis207_180 P3_IDPut <-> Device 3 (EtherCAT)/Box 2 (CU1128)/Term 24 (CU1128-B)/二维码胶拉胶[180] (InoSV660N)
//     Drive/Inputs/In/nDataIn1 <-> Inputs/Following error actual value
//     Drive/Inputs/In/nDataIn3[0] <-> Inputs/Torque actual value
//     Drive/Inputs/In/nDcOutputTime <-> InfoData/DcOutputShift
//     Drive/Inputs/In/nState1 <-> Inputs/Statusword
//     Drive/Inputs/In/nState2 <-> Inputs/Statusword @bit 8
//     Drive/Inputs/In/nState4 @bit 1 <-> WcState/InputToggle
//     Drive/Inputs/In/nState4 <-> WcState/WcState
//     Drive/Outputs/Out/nCtrl1 <-> Outputs/Controlword
//     Drive/Outputs/Out/nCtrl2 <-> Outputs/Controlword @bit 8
//     Drive/Outputs/Out/nDataOut1 <-> Outputs/Target position
//     Enc/Inputs/In/nDataIn1 <-> Inputs/Position actual value
//     Enc/Inputs/In/nDataIn3 <-> Inputs/Touch probe pos1 pos value
//     Enc/Inputs/In/nDataIn5 <-> Inputs/Touch probe pos2 pos value
//     Enc/Inputs/In/nDcInputTime <-> InfoData/DcInputShift
//     Enc/Inputs/In/nState4 @bit 1 <-> WcState/InputToggle
//     Enc/Inputs/In/nState4 <-> WcState/WcState
//     Enc/Inputs/In/nState5 <-> Inputs/Touch probe status
//     Enc/Inputs/In/nState6 <-> Inputs/Touch probe status @bit 8
//     Enc/Outputs/Out/nCtrl5 <-> Outputs/Touch probe function
//     Enc/Outputs/Out/nCtrl6 <-> Outputs/Touch probe function @bit 8
//   NC-Task 1 SAF/Axes/Axis208_181 P3_IDLift <-> Device 3 (EtherCAT)/Box 2 (CU1128)/Term 24 (CU1128-B)/二维码胶拉胶升降[181] (InoSV660N)
//     Drive/Inputs/In/nDataIn1 <-> Inputs/Following error actual value
//     Drive/Inputs/In/nDataIn3[0] <-> Inputs/Torque actual value
//     Drive/Inputs/In/nDcOutputTime <-> InfoData/DcOutputShift
//     Drive/Inputs/In/nState1 <-> Inputs/Statusword
//     Drive/Inputs/In/nState2 <-> Inputs/Statusword @bit 8
//     Drive/Inputs/In/nState4 @bit 1 <-> WcState/InputToggle
//     Drive/Inputs/In/nState4 <-> WcState/WcState
//     Drive/Outputs/Out/nCtrl1 <-> Outputs/Controlword
//     Drive/Outputs/Out/nCtrl2 <-> Outputs/Controlword @bit 8
//     Drive/Outputs/Out/nDataOut1 <-> Outputs/Target position
//     Enc/Inputs/In/nDataIn1 <-> Inputs/Position actual value
//     Enc/Inputs/In/nDataIn3 <-> Inputs/Touch probe pos1 pos value
//     Enc/Inputs/In/nDataIn5 <-> Inputs/Touch probe pos2 pos value
//     Enc/Inputs/In/nDcInputTime <-> InfoData/DcInputShift
//     Enc/Inputs/In/nState4 @bit 1 <-> WcState/InputToggle
//     Enc/Inputs/In/nState4 <-> WcState/WcState
//     Enc/Inputs/In/nState5 <-> Inputs/Touch probe status
//     Enc/Inputs/In/nState6 <-> Inputs/Touch probe status @bit 8
//     Enc/Outputs/Out/nCtrl5 <-> Outputs/Touch probe function
//     Enc/Outputs/Out/nCtrl6 <-> Outputs/Touch probe function @bit 8
//   DPPLC/DPPLC Instance <-> Device 3 (EtherCAT)/Box 2 (CU1128)/Box 61 (GSIO-A-SCU)
//     Task_P3 Inputs/P3IO.P3ShortReCrtl/InitAccepted <-> Module 34 (Free Port Mode COM2)/Inputs COM2/Status/Init accepted
//     Task_P3 Inputs/P3IO.P3ShortReCrtl/InputLength <-> Module 34 (Free Port Mode COM2)/Inputs COM2/Status/Input length
//     Task_P3 Inputs/P3IO.P3ShortReCrtl/PutDataDone <-> Module 34 (Free Port Mode COM2)/Inputs COM2/Status/PutData Done
//     Task_P3 Inputs/P3IO.P3ShortReCrtl/ReceiveRequest <-> Module 34 (Free Port Mode COM2)/Inputs COM2/Status/Receive request
//     Task_P3 Inputs/P3IO.P3ShortReCrtl/SndBufferFull <-> Module 34 (Free Port Mode COM2)/Inputs COM2/Status/SndBuffer full
//     Task_P3 Inputs/P3IO.P3ShortReCrtl/TotalInputLength <-> Module 34 (Free Port Mode COM2)/Inputs COM2/Status/Total input length
//     Task_P3 Inputs/P3IO.P3ShortReCrtl/TransmitDone <-> Module 34 (Free Port Mode COM2)/Inputs COM2/Status/Transmit Done
//     Task_P3 Inputs/P3IO.P3ShortTestRec.arrData[{1..32}] <-> Module 34 (Free Port Mode COM2)/Inputs COM2/Data In {0..31}  (32 links)
//     Task_P3 Inputs/P3IO.P3WeightRec.Data[{0..31}] <-> Module 33 (Free Port Mode COM1)/Inputs COM1/Data In {0..31}  (32 links)
//     Task_P3 Inputs/P3IO.P3WeightRec.Status/InitAccepted <-> Module 33 (Free Port Mode COM1)/Inputs COM1/Status/Init accepted
//     Task_P3 Inputs/P3IO.P3WeightRec.Status/InputLength <-> Module 33 (Free Port Mode COM1)/Inputs COM1/Status/Input length
//     Task_P3 Inputs/P3IO.P3WeightRec.Status/PutDataDone <-> Module 33 (Free Port Mode COM1)/Inputs COM1/Status/PutData Done
//     Task_P3 Inputs/P3IO.P3WeightRec.Status/ReceiveRequest <-> Module 33 (Free Port Mode COM1)/Inputs COM1/Status/Receive request
//     Task_P3 Inputs/P3IO.P3WeightRec.Status/SndBufferFull <-> Module 33 (Free Port Mode COM1)/Inputs COM1/Status/SndBuffer full
//     Task_P3 Inputs/P3IO.P3WeightRec.Status/TotalInputLength <-> Module 33 (Free Port Mode COM1)/Inputs COM1/Status/Total input length
//     Task_P3 Inputs/P3IO.P3WeightRec.Status/TransmitDone <-> Module 33 (Free Port Mode COM1)/Inputs COM1/Status/Transmit Done
//     Task_P3 Outputs/P3IO.P3ShortSendCrtl/InitRequest <-> Module 34 (Free Port Mode COM2)/Outputs COM2/Ctrl/Init request
//     Task_P3 Outputs/P3IO.P3ShortSendCrtl/OutputLength <-> Module 34 (Free Port Mode COM2)/Outputs COM2/Ctrl/Output length
//     Task_P3 Outputs/P3IO.P3ShortSendCrtl/PutData <-> Module 34 (Free Port Mode COM2)/Outputs COM2/Ctrl/Put data
//     Task_P3 Outputs/P3IO.P3ShortSendCrtl/ReceiveAccepted <-> Module 34 (Free Port Mode COM2)/Outputs COM2/Ctrl/Receive accepted
//     Task_P3 Outputs/P3IO.P3ShortSendCrtl/TransmitRequest <-> Module 34 (Free Port Mode COM2)/Outputs COM2/Ctrl/Transmit request
//     Task_P3 Outputs/P3IO.P3ShortTestSend.arrData[{1..32}] <-> Module 34 (Free Port Mode COM2)/Outputs COM2/Data Out {0..31}  (32 links)
//     Task_P3 Outputs/P3IO.P3WeightSend.Data[{0..31}] <-> Module 33 (Free Port Mode COM1)/Outputs COM1/Data Out {0..31}  (32 links)
//     Task_P3 Outputs/P3IO.P3WeightSend.Status/InitRequest <-> Module 33 (Free Port Mode COM1)/Outputs COM1/Ctrl/Init request
//     Task_P3 Outputs/P3IO.P3WeightSend.Status/OutputLength <-> Module 33 (Free Port Mode COM1)/Outputs COM1/Ctrl/Output length
//     Task_P3 Outputs/P3IO.P3WeightSend.Status/PutData <-> Module 33 (Free Port Mode COM1)/Outputs COM1/Ctrl/Put data
//     Task_P3 Outputs/P3IO.P3WeightSend.Status/ReceiveAccepted <-> Module 33 (Free Port Mode COM1)/Outputs COM1/Ctrl/Receive accepted
//     Task_P3 Outputs/P3IO.P3WeightSend.Status/TransmitRequest <-> Module 33 (Free Port Mode COM1)/Outputs COM1/Ctrl/Transmit request
//   DPPLC/DPPLC Instance <-> Device 3 (EtherCAT)/Box 2 (CU1128)/Box 68 (DL-EC1A)
//     Task_P3 Inputs/P3IO.ThicknessPar <-> ID01 Current Value/ID01 Current Value (P.V.)
//   DPPLC/DPPLC Instance <-> Device 3 (EtherCAT)/Box 2 (CU1128)/Term 24 (CU1128-B)/二维码胶拉胶[180] (InoSV660N)
//     Task_P2Main Inputs/GMotion.arrAxisCtrl[180].Io.DigitalInputs <-> Inputs/Digital inputs
//     Task_P2Main Inputs/IO.Network5_OP[17] <-> InfoData/State
//   DPPLC/DPPLC Instance <-> Device 3 (EtherCAT)/Box 2 (CU1128)/Term 24 (CU1128-B)/二维码胶拉胶升降[181] (InoSV660N)
//     Task_P2Main Inputs/GMotion.arrAxisCtrl[181].Io.DigitalInputs <-> Inputs/Digital inputs
//     Task_P2Main Inputs/IO.Network5_OP[18] <-> InfoData/State
//   DPPLC/DPPLC Instance <-> Device 3 (EtherCAT)/Box 2 (CU1128)/Term 24 (CU1128-B)/冷压托板开合[164] (CL3C-EC503)
//     Task_P2Main Inputs/GMotion.arrAxisCtrl[164].Io.DigitalInputs <-> Transmit PDO 1/Digital Inputs
//     Task_P2Main Inputs/IO.Network5_OP[14] <-> InfoData/State
//   DPPLC/DPPLC Instance <-> Device 3 (EtherCAT)/Box 2 (CU1128)/Term 24 (CU1128-B)/冷压驱动[165](InoSV660N)
//     Task_P2Main Inputs/GMotion.arrAxisCtrl[165].Io.DigitalInputs <-> Inputs/Digital inputs
//     Task_P2Main Inputs/GMotion.iActTorque_D[165] <-> Inputs/Torque actual value
//     Task_P2Main Inputs/IO.Network5_OP[9] <-> InfoData/State
//   DPPLC/DPPLC Instance <-> Device 3 (EtherCAT)/Box 2 (CU1128)/Term 24 (CU1128-B)/烤箱上料夹升降[168](InoSV660N)
//     Task_P2Main Inputs/GMotion.iActTorque_D[168] <-> Inputs/Torque actual value
//     Task_P2Main Inputs/IO.Network5_OP[3] <-> InfoData/State
//     Task_P3 Inputs/P3Motion.arrAxisCtrlV2[168].Io.DigitalInputs <-> Inputs/Digital inputs
//   DPPLC/DPPLC Instance <-> Device 3 (EtherCAT)/Box 2 (CU1128)/Term 24 (CU1128-B)/烤箱上料夹搬运[166] (InoSV660N)
//     Task_P2Main Inputs/GMotion.iActTorque_D[166] <-> Inputs/Torque actual value
//     Task_P2Main Inputs/IO.Network5_OP[2] <-> InfoData/State
//     Task_P3 Inputs/P3Motion.arrAxisCtrlV2[166].Io.DigitalInputs <-> Inputs/Digital inputs
//   DPPLC/DPPLC Instance <-> Device 3 (EtherCAT)/Box 2 (CU1128)/Term 24 (CU1128-B)/烤箱上料夹进退[167] (InoSV660N)
//     Task_P2Main Inputs/GMotion.iActTorque_D[167] <-> Inputs/Torque actual value
//     Task_P2Main Inputs/IO.Network5_OP[6] <-> InfoData/State
//     Task_P3 Inputs/P3Motion.arrAxisCtrlV2[167].Io.DigitalInputs <-> Inputs/Digital inputs
//   DPPLC/DPPLC Instance <-> Device 3 (EtherCAT)/Box 2 (CU1128)/Term 24 (CU1128-B)/热压托板开合[169] (CL3C-EC503)
//     Task_P2Main Inputs/GMotion.arrAxisCtrl[169].Io.DigitalInputs <-> Transmit PDO 1/Digital Inputs
//     Task_P2Main Inputs/IO.Network5_OP[7] <-> InfoData/State
//   DPPLC/DPPLC Instance <-> Device 3 (EtherCAT)/Box 2 (CU1128)/Term 24 (CU1128-B)/热压驱动[170] (InoSV660N)
//     Task_P2Main Inputs/GMotion.arrAxisCtrl[170].Io.DigitalInputs <-> Inputs/Digital inputs
//     Task_P2Main Inputs/GMotion.iActTorque_D[170] <-> Inputs/Torque actual value
//     Task_P2Main Inputs/IO.Network5_OP[8] <-> InfoData/State
//   DPPLC/DPPLC Instance <-> Device 3 (EtherCAT)/Box 2 (CU1128)/Term 24 (CU1128-B)/电芯下料夹升降[177] (InoSV660N)
//     Task_P2Main Inputs/GMotion.arrAxisCtrl[177].Io.DigitalInputs <-> Inputs/Digital inputs
//     Task_P2Main Inputs/GMotion.iActTorque_D[177] <-> Inputs/Torque actual value
//     Task_P2Main Inputs/IO.Network5_OP[12] <-> InfoData/State
//   DPPLC/DPPLC Instance <-> Device 3 (EtherCAT)/Box 2 (CU1128)/Term 24 (CU1128-B)/电芯下料夹搬运[176] (InoSV660N)
//     Task_P2Main Inputs/GMotion.arrAxisCtrl[176].Io.DigitalInputs <-> Inputs/Digital inputs
//     Task_P2Main Inputs/GMotion.iActTorque_D[176] <-> Inputs/Torque actual value
//     Task_P2Main Inputs/IO.Network5_OP[11] <-> InfoData/State
//   DPPLC/DPPLC Instance <-> Device 3 (EtherCAT)/Box 2 (CU1128)/Term 24 (CU1128-B)/电芯分选夹升降[175] (InoSV660N)
//     Task_P2Main Inputs/GMotion.arrAxisCtrl[175].Io.DigitalInputs <-> Inputs/Digital inputs
//     Task_P2Main Inputs/GMotion.iActTorque_D[175] <-> Inputs/Torque actual value
//     Task_P2Main Inputs/IO.Network5_OP[13] <-> InfoData/State
//   DPPLC/DPPLC Instance <-> Device 3 (EtherCAT)/Box 2 (CU1128)/Term 24 (CU1128-B)/电芯分选夹搬运[174](InoSV660N)
//     Task_P2Main Inputs/GMotion.arrAxisCtrl[174].Io.DigitalInputs <-> Inputs/Digital inputs
//     Task_P2Main Inputs/GMotion.iActTorque_D[174] <-> Inputs/Torque actual value
//     Task_P2Main Inputs/IO.Network5_OP[10] <-> InfoData/State
//   DPPLC/DPPLC Instance <-> Device 3 (EtherCAT)/Box 2 (CU1128)/Term 24 (CU1128-B)/称重上料夹升降[172](InoSV660N)
//     Task_P2Main Inputs/GMotion.arrAxisCtrl[172].Io.DigitalInputs <-> Inputs/Digital inputs
//     Task_P2Main Inputs/GMotion.iActTorque_D[172] <-> Inputs/Torque actual value
//     Task_P2Main Inputs/IO.Network5_OP[4] <-> InfoData/State
//   DPPLC/DPPLC Instance <-> Device 3 (EtherCAT)/Box 2 (CU1128)/Term 24 (CU1128-B)/称重上料夹平移[171] (InoSV660N)
//     Task_P2Main Inputs/GMotion.arrAxisCtrl[171].Io.DigitalInputs <-> Inputs/Digital inputs
//     Task_P2Main Inputs/GMotion.iActTorque_D[171] <-> Inputs/Torque actual value
//     Task_P2Main Inputs/IO.Network5_OP[1] <-> InfoData/State
//   DPPLC/DPPLC Instance <-> Device 3 (EtherCAT)/Box 2 (CU1128)/Term 24 (CU1128-B)/称重上料夹旋转[173] (InoSV660N)
//     Task_P2Main Inputs/GMotion.arrAxisCtrl[173].Io.DigitalInputs <-> Inputs/Digital inputs
//     Task_P2Main Inputs/GMotion.iActTorque_D[173] <-> Inputs/Torque actual value
//     Task_P2Main Inputs/IO.Network5_OP[5] <-> InfoData/State
//   DPPLC/DPPLC Instance <-> Device 3 (EtherCAT)/Box 2 (CU1128)/Term 24 (CU1128-B)/贴胶头进退 [178](InoSV660N)
//     Task_P2Main Inputs/GMotion.arrAxisCtrl[178].Io.DigitalInputs <-> Inputs/Digital inputs
//     Task_P2Main Inputs/GMotion.iActTorque_D[178] <-> Inputs/Torque actual value
//     Task_P2Main Inputs/IO.Network5_OP[15] <-> InfoData/State
//   DPPLC/DPPLC Instance <-> Device 3 (EtherCAT)/Box 2 (CU1128)/Term 24 (CU1128-B)/贴胶平移[179](InoSV660N)
//     Task_P2Main Inputs/GMotion.arrAxisCtrl[179].Io.DigitalInputs <-> Inputs/Digital inputs
//     Task_P2Main Inputs/GMotion.iActTorque_D[179] <-> Inputs/Torque actual value
//     Task_P2Main Inputs/IO.Network5_OP[16] <-> InfoData/State
//   DPPLC/DPPLC Instance <-> Device 3 (EtherCAT)/Box 2 (CU1128)/Term 44 (CU1128-C)/P2M2M隔膜放卷纠偏[67] (InoSV660N)
//     Task_P2Main Inputs/GMotion.arrAxisCtrl[67].Io.DigitalInputs <-> Inputs/Digital inputs
//     Task_P2Main Inputs/GMotion.iActTorque_D[67] <-> Inputs/Torque actual value
//     Task_P2Main Inputs/IO.Network2_OP[2] <-> InfoData/State
//   DPPLC/DPPLC Instance <-> Device 3 (EtherCAT)/Box 2 (CU1128)/Term 44 (CU1128-C)/P2M2侧贴夹平移[87] (InoSV660N)
//     Task_P2Main Inputs/GMotion.arrAxisCtrl[87].Io.DigitalInputs <-> Inputs/Digital inputs
//     Task_P2Main Inputs/GMotion.iActTorque_D[87] <-> Inputs/Torque actual value
//     Task_P2Main Inputs/IO.Network2_OP[24] <-> InfoData/State
//   DPPLC/DPPLC Instance <-> Device 3 (EtherCAT)/Box 2 (CU1128)/Term 44 (CU1128-C)/P2M2侧贴夹旋转 [88](InoSV660N)
//     Task_P2Main Inputs/GMotion.arrAxisCtrl[88].Io.DigitalInputs <-> Inputs/Digital inputs
//     Task_P2Main Inputs/GMotion.iActTorque_D[88] <-> Inputs/Torque actual value
//     Task_P2Main Inputs/IO.Network2_OP[25] <-> InfoData/State
//   DPPLC/DPPLC Instance <-> Device 3 (EtherCAT)/Box 2 (CU1128)/Term 44 (CU1128-C)/P2M2冷压上料夹升降[163（热压）] (InoSV660N)
//     Task_P2Main Inputs/GMotion.arrAxisCtrl[163].Io.DigitalInputs <-> Inputs/Digital inputs
//     Task_P2Main Inputs/GMotion.iActTorque_D[163] <-> Inputs/Torque actual value
//     Task_P2Main Inputs/IO.Network2_OP[49] <-> InfoData/State
//   DPPLC/DPPLC Instance <-> Device 3 (EtherCAT)/Box 2 (CU1128)/Term 44 (CU1128-C)/P2M2冷压上料夹旋转[162（热压）] (InoSV660N)
//     Task_P2Main Inputs/GMotion.arrAxisCtrl[162].Io.DigitalInputs <-> Inputs/Digital inputs
//     Task_P2Main Inputs/GMotion.iActTorque_D[162] <-> Inputs/Torque actual value
//     Task_P2Main Inputs/IO.Network2_OP[48] <-> InfoData/State
//   DPPLC/DPPLC Instance <-> Device 3 (EtherCAT)/Box 2 (CU1128)/Term 44 (CU1128-C)/P2M2冷压上料夹进退[161（热压）] (InoSV660N)
//     Task_P2Main Inputs/GMotion.arrAxisCtrl[161].Io.DigitalInputs <-> Inputs/Digital inputs
//     Task_P2Main Inputs/GMotion.iActTorque_D[161] <-> Inputs/Torque actual value
//     Task_P2Main Inputs/IO.Network2_OP[47] <-> InfoData/State
//   DPPLC/DPPLC Instance <-> Device 3 (EtherCAT)/Box 2 (CU1128)/Term 44 (CU1128-C)/P2M2叠台升降[72] (InoSV660N)
//     Task_P2Main Inputs/GMotion.arrAxisCtrl[72].Io.DigitalInputs <-> Inputs/Digital inputs
//     Task_P2Main Inputs/GMotion.iActTorque_D[72] <-> Inputs/Torque actual value
//     Task_P2Main Inputs/IO.Network2_OP[38] <-> InfoData/State
//   DPPLC/DPPLC Instance <-> Device 3 (EtherCAT)/Box 2 (CU1128)/Term 44 (CU1128-C)/P2M2右压刀升降[76] (InoSV660N)
//     Task_P2Main Inputs/GMotion.arrAxisCtrl[76].Io.DigitalInputs <-> Inputs/Digital inputs
//     Task_P2Main Inputs/GMotion.iActTorque_D[76] <-> Inputs/Torque actual value
//     Task_P2Main Inputs/IO.Network2_OP[42] <-> InfoData/State
//   DPPLC/DPPLC Instance <-> Device 3 (EtherCAT)/Box 2 (CU1128)/Term 44 (CU1128-C)/P2M2右压刀开合[75] (InoSV660N)
//     Task_P2Main Inputs/GMotion.arrAxisCtrl[75].Io.DigitalInputs <-> Inputs/Digital inputs
//     Task_P2Main Inputs/GMotion.iActTorque_D[75] <-> Inputs/Torque actual value
//     Task_P2Main Inputs/IO.Network2_OP[41] <-> InfoData/State
//   DPPLC/DPPLC Instance <-> Device 3 (EtherCAT)/Box 2 (CU1128)/Term 44 (CU1128-C)/P2M2夹膜升降 [82](InoSV660N)
//     Task_P2Main Inputs/GMotion.arrAxisCtrl[82].Io.DigitalInputs <-> Inputs/Digital inputs
//     Task_P2Main Inputs/GMotion.iActTorque_D[82] <-> Inputs/Torque actual value
//     Task_P2Main Inputs/IO.Network2_OP[23] <-> InfoData/State
//   DPPLC/DPPLC Instance <-> Device 3 (EtherCAT)/Box 2 (CU1128)/Term 44 (CU1128-C)/P2M2夹膜平移[81] (InoSV660N)
//     Task_P2Main Inputs/GMotion.arrAxisCtrl[81].Io.DigitalInputs <-> Inputs/Digital inputs
//     Task_P2Main Inputs/GMotion.iActTorque_D[81] <-> Inputs/Torque actual value
//     Task_P2Main Inputs/IO.Network2_OP[22] <-> InfoData/State
//   DPPLC/DPPLC Instance <-> Device 3 (EtherCAT)/Box 2 (CU1128)/Term 44 (CU1128-C)/P2M2尾卷夹电芯伸缩[79] (InoSV660N)
//     Task_P2Main Inputs/GMotion.arrAxisCtrl[79].Io.DigitalInputs <-> Inputs/Digital inputs
//     Task_P2Main Inputs/GMotion.iActTorque_D[79] <-> Inputs/Torque actual value
//     Task_P2Main Inputs/IO.Network2_OP[20] <-> InfoData/State
//   DPPLC/DPPLC Instance <-> Device 3 (EtherCAT)/Box 2 (CU1128)/Term 44 (CU1128-C)/P2M2尾卷夹电芯升降[78] (InoSV660N)
//     Task_P2Main Inputs/GMotion.arrAxisCtrl[78].Io.DigitalInputs <-> Inputs/Digital inputs
//     Task_P2Main Inputs/GMotion.iActTorque_D[78] <-> Inputs/Torque actual value
//     Task_P2Main Inputs/IO.Network2_OP[19] <-> InfoData/State
//   DPPLC/DPPLC Instance <-> Device 3 (EtherCAT)/Box 2 (CU1128)/Term 44 (CU1128-C)/P2M2尾卷夹电芯平移[77] (InoSV660N)
//     Task_P2Main Inputs/GMotion.arrAxisCtrl[77].Io.DigitalInputs <-> Inputs/Digital inputs
//     Task_P2Main Inputs/GMotion.iActTorque_D[77] <-> Inputs/Torque actual value
//     Task_P2Main Inputs/IO.Network2_OP[18] <-> InfoData/State
//   DPPLC/DPPLC Instance <-> Device 3 (EtherCAT)/Box 2 (CU1128)/Term 44 (CU1128-C)/P2M2尾卷夹电芯旋转[80](InoSV660N)
//     Task_P2Main Inputs/GMotion.arrAxisCtrl[80].Io.DigitalInputs <-> Inputs/Digital inputs
//     Task_P2Main Inputs/GMotion.iActTorque_D[80] <-> Inputs/Torque actual value
//     Task_P2Main Inputs/IO.Network2_OP[21] <-> InfoData/State
//   DPPLC/DPPLC Instance <-> Device 3 (EtherCAT)/Box 2 (CU1128)/Term 44 (CU1128-C)/P2M2左压刀升降[74] (InoSV660N)
//     Task_P2Main Inputs/GMotion.arrAxisCtrl[74].Io.DigitalInputs <-> Inputs/Digital inputs
//     Task_P2Main Inputs/GMotion.iActTorque_D[74] <-> Inputs/Torque actual value
//     Task_P2Main Inputs/IO.Network2_OP[40] <-> InfoData/State
//   DPPLC/DPPLC Instance <-> Device 3 (EtherCAT)/Box 2 (CU1128)/Term 44 (CU1128-C)/P2M2左压刀开合[73](InoSV660N)
//     Task_P2Main Inputs/GMotion.arrAxisCtrl[73].Io.DigitalInputs <-> Inputs/Digital inputs
//     Task_P2Main Inputs/GMotion.iActTorque_D[73] <-> Inputs/Torque actual value
//     Task_P2Main Inputs/IO.Network2_OP[39] <-> InfoData/State
//   DPPLC/DPPLC Instance <-> Device 3 (EtherCAT)/Box 2 (CU1128)/Term 44 (CU1128-C)/P2M2拉胶升降 [90](InoSV660N)
//     Task_P2Main Inputs/GMotion.arrAxisCtrl[90].Io.DigitalInputs <-> Inputs/Digital inputs
//     Task_P2Main Inputs/GMotion.iActTorque_D[90] <-> Inputs/Torque actual value
//     Task_P2Main Inputs/IO.Network2_OP[33] <-> InfoData/State
//   DPPLC/DPPLC Instance <-> Device 3 (EtherCAT)/Box 2 (CU1128)/Term 44 (CU1128-C)/P2M2正极叠台搬运升降[51] (InoSV660N)
//     Task_P2Main Inputs/GMotion.arrAxisCtrl[51].Io.DigitalInputs <-> Inputs/Digital inputs
//     Task_P2Main Inputs/GMotion.iActTorque_D[51] <-> Inputs/Torque actual value
//     Task_P2Main Inputs/IO.Network2_OP[7] <-> InfoData/State
//   DPPLC/DPPLC Instance <-> Device 3 (EtherCAT)/Box 2 (CU1128)/Term 44 (CU1128-C)/P2M2正极叠台搬运平移1[50](CDHD)
//     Task_P2Main Inputs/GMotion.arrAxisCtrl[50].Io.DigitalInputs <-> TxPDO 4/Digital inputs
//     Task_P2Main Inputs/GMotion.iActTorque_D[50] <-> TxPDO 1/Torque Actual Value
//     Task_P2Main Inputs/IO.Network2_OP[11] <-> InfoData/State
//   DPPLC/DPPLC Instance <-> Device 3 (EtherCAT)/Box 2 (CU1128)/Term 44 (CU1128-C)/P2M2正极纠偏平台X1[52] (InoSV660N)
//     Task_P2Main Inputs/GMotion.arrAxisCtrl[52].Io.DigitalInputs <-> Inputs/Digital inputs
//     Task_P2Main Inputs/GMotion.iActTorque_D[52] <-> Inputs/Torque actual value
//     Task_P2Main Inputs/IO.Network2_OP[9] <-> InfoData/State
//   DPPLC/DPPLC Instance <-> Device 3 (EtherCAT)/Box 2 (CU1128)/Term 44 (CU1128-C)/P2M2正极纠偏平台X2[53](InoSV660N)
//     Task_P2Main Inputs/GMotion.arrAxisCtrl[53].Io.DigitalInputs <-> Inputs/Digital inputs
//     Task_P2Main Inputs/GMotion.iActTorque_D[53] <-> Inputs/Torque actual value
//     Task_P2Main Inputs/IO.Network2_OP[14] <-> InfoData/State
//   DPPLC/DPPLC Instance <-> Device 3 (EtherCAT)/Box 2 (CU1128)/Term 44 (CU1128-C)/P2M2正极纠偏平台Y[54] (InoSV660N)
//     Task_P2Main Inputs/GMotion.arrAxisCtrl[54].Io.DigitalInputs <-> Inputs/Digital inputs
//     Task_P2Main Inputs/GMotion.iActTorque_D[54] <-> Inputs/Torque actual value
//     Task_P2Main Inputs/IO.Network2_OP[15] <-> InfoData/State
//   DPPLC/DPPLC Instance <-> Device 3 (EtherCAT)/Box 2 (CU1128)/Term 44 (CU1128-C)/P2M2正极送料分段皮带2[21(模切)] (InoSV660N)
//     Task_P2Main Inputs/IO.Network2_OP[1] <-> InfoData/State
//   DPPLC/DPPLC Instance <-> Device 3 (EtherCAT)/Box 2 (CU1128)/Term 44 (CU1128-C)/P2M2正极送片搬运升降[48] (InoSV660N)
//     Task_P2Main Inputs/GMotion.arrAxisCtrl[48].Io.DigitalInputs <-> Inputs/Digital inputs
//     Task_P2Main Inputs/GMotion.iActTorque_D[48] <-> Inputs/Torque actual value
//     Task_P2Main Inputs/IO.Network2_OP[5] <-> InfoData/State
//   DPPLC/DPPLC Instance <-> Device 3 (EtherCAT)/Box 2 (CU1128)/Term 44 (CU1128-C)/P2M2正极送片搬运平移 [47](CDHD)
//     Task_P2Main Inputs/GMotion.arrAxisCtrl[47].Io.DigitalInputs <-> TxPDO 4/Digital inputs
//     Task_P2Main Inputs/GMotion.iActTorque_D[47] <-> TxPDO 1/Torque Actual Value
//     Task_P2Main Inputs/IO.Network2_OP[10] <-> InfoData/State
//   DPPLC/DPPLC Instance <-> Device 3 (EtherCAT)/Box 2 (CU1128)/Term 44 (CU1128-C)/P2M2正极送片搬运旋转[49] (InoSV660N)
//     Task_P2Main Inputs/GMotion.arrAxisCtrl[49].Io.DigitalInputs <-> Inputs/Digital inputs
//     Task_P2Main Inputs/GMotion.iActTorque_D[49] <-> Inputs/Torque actual value
//     Task_P2Main Inputs/IO.Network2_OP[6] <-> InfoData/State
//   DPPLC/DPPLC Instance <-> Device 3 (EtherCAT)/Box 2 (CU1128)/Term 44 (CU1128-C)/P2M2短卷针平移[84](CL3C-EC808AC)
//     Task_P2Main Inputs/GMotion.arrAxisCtrl[84].Io.DigitalInputs <-> Transmit PDO 1/Digital Inputs
//     Task_P2Main Inputs/IO.Network2_OP[35] <-> InfoData/State
//   DPPLC/DPPLC Instance <-> Device 3 (EtherCAT)/Box 2 (CU1128)/Term 44 (CU1128-C)/P2M2短卷针旋转[86] (CL3C-EC808AC)
//     Task_P2Main Inputs/GMotion.arrAxisCtrl[86].Io.DigitalInputs <-> Transmit PDO 1/Digital Inputs
//     Task_P2Main Inputs/IO.Network2_OP[37] <-> InfoData/State
//   DPPLC/DPPLC Instance <-> Device 3 (EtherCAT)/Box 2 (CU1128)/Term 44 (CU1128-C)/P2M2负极叠台搬运升降 [62](InoSV660N)
//     Task_P2Main Inputs/GMotion.arrAxisCtrl[62].Io.DigitalInputs <-> Inputs/Digital inputs
//     Task_P2Main Inputs/GMotion.iActTorque_D[62] <-> Inputs/Torque actual value
//     Task_P2Main Inputs/IO.Network2_OP[46] <-> InfoData/State
//   DPPLC/DPPLC Instance <-> Device 3 (EtherCAT)/Box 2 (CU1128)/Term 44 (CU1128-C)/P2M2负极叠台搬运平移[61](CDHD)
//     Task_P2Main Inputs/GMotion.arrAxisCtrl[61].Io.DigitalInputs <-> TxPDO 4/Digital inputs
//     Task_P2Main Inputs/GMotion.iActTorque_D[61] <-> TxPDO 1/Torque Actual Value
//     Task_P2Main Inputs/IO.Network2_OP[29] <-> InfoData/State
//   DPPLC/DPPLC Instance <-> Device 3 (EtherCAT)/Box 2 (CU1128)/Term 44 (CU1128-C)/P2M2负极纠偏平台X1 [63](InoSV660N)
//     Task_P2Main Inputs/GMotion.arrAxisCtrl[63].Io.DigitalInputs <-> Inputs/Digital inputs
//     Task_P2Main Inputs/GMotion.iActTorque_D[63] <-> Inputs/Torque actual value
//     Task_P2Main Inputs/IO.Network2_OP[30] <-> InfoData/State
//   DPPLC/DPPLC Instance <-> Device 3 (EtherCAT)/Box 2 (CU1128)/Term 44 (CU1128-C)/P2M2负极纠偏平台X2[64] (InoSV660N)
//     Task_P2Main Inputs/GMotion.arrAxisCtrl[64].Io.DigitalInputs <-> Inputs/Digital inputs
//     Task_P2Main Inputs/GMotion.iActTorque_D[64] <-> Inputs/Torque actual value
//     Task_P2Main Inputs/IO.Network2_OP[31] <-> InfoData/State
//   DPPLC/DPPLC Instance <-> Device 3 (EtherCAT)/Box 2 (CU1128)/Term 44 (CU1128-C)/P2M2负极纠偏平台Y[65](InoSV660N)
//     Task_P2Main Inputs/GMotion.arrAxisCtrl[65].Io.DigitalInputs <-> Inputs/Digital inputs
//     Task_P2Main Inputs/GMotion.iActTorque_D[65] <-> Inputs/Torque actual value
//     Task_P2Main Inputs/IO.Network2_OP[32] <-> InfoData/State
//   DPPLC/DPPLC Instance <-> Device 3 (EtherCAT)/Box 2 (CU1128)/Term 44 (CU1128-C)/P2M2负极送料分段皮带2（45模切） (InoSV660N)
//     Task_P2Main Inputs/IO.Network2_OP[16] <-> InfoData/State
//   DPPLC/DPPLC Instance <-> Device 3 (EtherCAT)/Box 2 (CU1128)/Term 44 (CU1128-C)/P2M2负极送片搬运1升降[56] (InoSV660N)
//     Task_P2Main Inputs/GMotion.arrAxisCtrl[56].Io.DigitalInputs <-> Inputs/Digital inputs
//     Task_P2Main Inputs/GMotion.iActTorque_D[56] <-> Inputs/Torque actual value
//     Task_P2Main Inputs/IO.Network2_OP[43] <-> InfoData/State
//   DPPLC/DPPLC Instance <-> Device 3 (EtherCAT)/Box 2 (CU1128)/Term 44 (CU1128-C)/P2M2负极送片搬运1平移[55] (CDHD)
//     Task_P2Main Inputs/GMotion.arrAxisCtrl[55].Io.DigitalInputs <-> TxPDO 4/Digital inputs
//     Task_P2Main Inputs/GMotion.iActTorque_D[55] <-> TxPDO 1/Torque Actual Value
//     Task_P2Main Inputs/IO.Network2_OP[27] <-> InfoData/State
//   DPPLC/DPPLC Instance <-> Device 3 (EtherCAT)/Box 2 (CU1128)/Term 44 (CU1128-C)/P2M2负极送片搬运1旋转 [57](InoSV660N)
//     Task_P2Main Inputs/GMotion.arrAxisCtrl[57].Io.DigitalInputs <-> Inputs/Digital inputs
//     Task_P2Main Inputs/GMotion.iActTorque_D[57] <-> Inputs/Torque actual value
//     Task_P2Main Inputs/IO.Network2_OP[44] <-> InfoData/State
//   DPPLC/DPPLC Instance <-> Device 3 (EtherCAT)/Box 2 (CU1128)/Term 44 (CU1128-C)/P2M2负极送片搬运2升降[59] (InoSV660N)
//     Task_P2Main Inputs/GMotion.arrAxisCtrl[59].Io.DigitalInputs <-> Inputs/Digital inputs
//     Task_P2Main Inputs/GMotion.iActTorque_D[59] <-> Inputs/Torque actual value
//     Task_P2Main Inputs/IO.Network2_OP[45] <-> InfoData/State
//   DPPLC/DPPLC Instance <-> Device 3 (EtherCAT)/Box 2 (CU1128)/Term 44 (CU1128-C)/P2M2负极送片搬运2平移[58] (CDHD)
//     Task_P2Main Inputs/GMotion.arrAxisCtrl[58].Io.DigitalInputs <-> TxPDO 4/Digital inputs
//     Task_P2Main Inputs/GMotion.iActTorque_D[58] <-> TxPDO 1/Torque Actual Value
//     Task_P2Main Inputs/IO.Network2_OP[28] <-> InfoData/State
//   DPPLC/DPPLC Instance <-> Device 3 (EtherCAT)/Box 2 (CU1128)/Term 44 (CU1128-C)/P2M2负极送片皮带[60](InoSV660N)
//     Task_P2Main Inputs/GMotion.arrAxisCtrl[60].Io.DigitalInputs <-> Inputs/Digital inputs
//     Task_P2Main Inputs/GMotion.iActTorque_D[60] <-> Inputs/Torque actual value
//     Task_P2Main Inputs/IO.Network2_OP[17] <-> InfoData/State
//   DPPLC/DPPLC Instance <-> Device 3 (EtherCAT)/Box 2 (CU1128)/Term 44 (CU1128-C)/P2M2贴胶头进退[89](InoSV660N)
//     Task_P2Main Inputs/GMotion.arrAxisCtrl[89].Io.DigitalInputs <-> Inputs/Digital inputs
//     Task_P2Main Inputs/GMotion.iActTorque_D[89] <-> Inputs/Torque actual value
//     Task_P2Main Inputs/IO.Network2_OP[26] <-> InfoData/State
//   DPPLC/DPPLC Instance <-> Device 3 (EtherCAT)/Box 2 (CU1128)/Term 44 (CU1128-C)/P2M2长卷针平移[83] (CL3C-EC808AC)
//     Task_P2Main Inputs/GMotion.arrAxisCtrl[83].Io.DigitalInputs <-> Transmit PDO 1/Digital Inputs
//     Task_P2Main Inputs/IO.Network2_OP[34] <-> InfoData/State
//   DPPLC/DPPLC Instance <-> Device 3 (EtherCAT)/Box 2 (CU1128)/Term 44 (CU1128-C)/P2M2长卷针旋转[85](CL3C-EC808AC)
//     Task_P2Main Inputs/GMotion.arrAxisCtrl[85].Io.DigitalInputs <-> Transmit PDO 1/Digital Inputs
//     Task_P2Main Inputs/IO.Network2_OP[36] <-> InfoData/State
//   DPPLC/DPPLC Instance <-> Device 3 (EtherCAT)/Box 2 (CU1128)/Term 44 (CU1128-C)/P2M2隔膜尾部纠偏[68] (InoSV660N)
//     Task_P2Main Inputs/GMotion.arrAxisCtrl[68].Io.DigitalInputs <-> Inputs/Digital inputs
//     Task_P2Main Inputs/GMotion.iActTorque_D[68] <-> Inputs/Torque actual value
//     Task_P2Main Inputs/IO.Network2_OP[8] <-> InfoData/State
//   DPPLC/DPPLC Instance <-> Device 3 (EtherCAT)/Box 2 (CU1128)/Term 44 (CU1128-C)/P2M2隔膜平移[71] (CDHD)
//     Task_P2Main Inputs/GMotion.arrAxisCtrl[71].Io.DigitalInputs <-> TxPDO 4/Digital inputs
//     Task_P2Main Inputs/GMotion.iActTorque_D[71] <-> TxPDO 1/Torque Actual Value
//     Task_P2Main Inputs/IO.Network2_OP[12] <-> InfoData/State
//   DPPLC/DPPLC Instance <-> Device 3 (EtherCAT)/Box 2 (CU1128)/Term 44 (CU1128-C)/P2M2隔膜摆杆张力[69](InoSV660N)
//     Task_P2M3 Outputs/GMotion.iTargetTorque[2] <-> Outputs/Target torque
//     Task_P2Main Inputs/GMotion.arrAxisCtrl[69].Io.DigitalInputs <-> Inputs/Digital inputs
//     Task_P2Main Inputs/GMotion.iActTorque_D[69] <-> Inputs/Torque actual value
//     Task_P2Main Inputs/IO.Network2_OP[3] <-> InfoData/State
//     Task_P3 Outputs/GMotion.iMaxProfileVelo[2] <-> Outputs/Max profile velocity
//     Task_P3 Outputs/GMotion.iNegtiveTorqueLimits[2] <-> Outputs/Negative torque limit value
//     Task_P3 Outputs/GMotion.iPostiveTorqueLimits[2] <-> Outputs/Positive torque limit value
//     Task_P3 Outputs/GMotion.iSetDriveMode[2] <-> Outputs/Modes of operation
//   DPPLC/DPPLC Instance <-> Device 3 (EtherCAT)/Box 2 (CU1128)/Term 44 (CU1128-C)/P2M2隔膜放卷[66](InoSV660N)
//     Task_P2Main Inputs/GMotion.arrAxisCtrl[66].Io.DigitalInputs <-> Inputs/Digital inputs
//     Task_P2Main Inputs/GMotion.iActTorque_D[66] <-> Inputs/Torque actual value
//     Task_P2Main Inputs/IO.Network2_OP[4] <-> InfoData/State
//   DPPLC/DPPLC Instance <-> Device 3 (EtherCAT)/Box 2 (CU1128)/Term 44 (CU1128-C)/P2M2隔膜缓存[70](CDHD)
//     Task_P2Main Inputs/GMotion.arrAxisCtrl[70].Io.DigitalInputs <-> TxPDO 4/Digital inputs
//     Task_P2Main Inputs/GMotion.iActTorque_D[70] <-> TxPDO 1/Torque Actual Value
//     Task_P2Main Inputs/IO.Network2_OP[13] <-> InfoData/State
//   DPPLC/DPPLC Instance <-> Device 3 (EtherCAT)/Box 2 (CU1128)/Term 44 (CU1128-C)/P2M3侧贴夹平移（ 133）(InoSV660N)
//     Task_P2Main Inputs/GMotion.arrAxisCtrl[133].Io.DigitalInputs <-> Inputs/Digital inputs
//     Task_P2Main Inputs/GMotion.iActTorque_D[133] <-> Inputs/Torque actual value
//     Task_P2Main Inputs/IO.Network3_OP[24] <-> InfoData/State
//   DPPLC/DPPLC Instance <-> Device 3 (EtherCAT)/Box 2 (CU1128)/Term 44 (CU1128-C)/P2M3侧贴夹旋转[134] (InoSV660N)
//     Task_P2Main Inputs/GMotion.arrAxisCtrl[134].Io.DigitalInputs <-> Inputs/Digital inputs
//     Task_P2Main Inputs/GMotion.iActTorque_D[134] <-> Inputs/Torque actual value
//     Task_P2Main Inputs/IO.Network3_OP[25] <-> InfoData/State
//   DPPLC/DPPLC Instance <-> Device 3 (EtherCAT)/Box 2 (CU1128)/Term 44 (CU1128-C)/P2M3叠台升降 [118](InoSV660N)
//     Task_P2Main Inputs/GMotion.arrAxisCtrl[118].Io.DigitalInputs <-> Inputs/Digital inputs
//     Task_P2Main Inputs/GMotion.iActTorque_D[118] <-> Inputs/Torque actual value
//     Task_P2Main Inputs/IO.Network3_OP[37] <-> InfoData/State
//   DPPLC/DPPLC Instance <-> Device 3 (EtherCAT)/Box 2 (CU1128)/Term 44 (CU1128-C)/P2M3右压刀升降 [122](InoSV660N)
//     Task_P2Main Inputs/GMotion.arrAxisCtrl[122].Io.DigitalInputs <-> Inputs/Digital inputs
//     Task_P2Main Inputs/GMotion.iActTorque_D[122] <-> Inputs/Torque actual value
//     Task_P2Main Inputs/IO.Network3_OP[41] <-> InfoData/State
//   DPPLC/DPPLC Instance <-> Device 3 (EtherCAT)/Box 2 (CU1128)/Term 44 (CU1128-C)/P2M3右压刀开合[121](InoSV660N)
//     Task_P2Main Inputs/GMotion.arrAxisCtrl[121].Io.DigitalInputs <-> Inputs/Digital inputs
//     Task_P2Main Inputs/GMotion.iActTorque_D[121] <-> Inputs/Torque actual value
//     Task_P2Main Inputs/IO.Network3_OP[40] <-> InfoData/State
//   DPPLC/DPPLC Instance <-> Device 3 (EtherCAT)/Box 2 (CU1128)/Term 44 (CU1128-C)/P2M3夹膜升降（128） (InoSV660N)
//     Task_P2Main Inputs/GMotion.arrAxisCtrl[128].Io.DigitalInputs <-> Inputs/Digital inputs
//     Task_P2Main Inputs/GMotion.iActTorque_D[128] <-> Inputs/Torque actual value
//     Task_P2Main Inputs/IO.Network3_OP[23] <-> InfoData/State
//   DPPLC/DPPLC Instance <-> Device 3 (EtherCAT)/Box 2 (CU1128)/Term 44 (CU1128-C)/P2M3夹膜平移 （127）(InoSV660N)
//     Task_P2Main Inputs/GMotion.arrAxisCtrl[127].Io.DigitalInputs <-> Inputs/Digital inputs
//     Task_P2Main Inputs/GMotion.iActTorque_D[127] <-> Inputs/Torque actual value
//     Task_P2Main Inputs/IO.Network3_OP[22] <-> InfoData/State
//   DPPLC/DPPLC Instance <-> Device 3 (EtherCAT)/Box 2 (CU1128)/Term 44 (CU1128-C)/P2M3尾卷夹电芯伸缩 （125）(InoSV660N)
//     Task_P2Main Inputs/GMotion.arrAxisCtrl[125].Io.DigitalInputs <-> Inputs/Digital inputs
//     Task_P2Main Inputs/GMotion.iActTorque_D[125] <-> Inputs/Torque actual value
//     Task_P2Main Inputs/IO.Network3_OP[20] <-> InfoData/State
//   DPPLC/DPPLC Instance <-> Device 3 (EtherCAT)/Box 2 (CU1128)/Term 44 (CU1128-C)/P2M3尾卷夹电芯升降（124） (InoSV660N)
//     Task_P2Main Inputs/GMotion.arrAxisCtrl[124].Io.DigitalInputs <-> Inputs/Digital inputs
//     Task_P2Main Inputs/GMotion.iActTorque_D[124] <-> Inputs/Torque actual value
//     Task_P2Main Inputs/IO.Network3_OP[19] <-> InfoData/State
//   DPPLC/DPPLC Instance <-> Device 3 (EtherCAT)/Box 2 (CU1128)/Term 44 (CU1128-C)/P2M3尾卷夹电芯平移（123） (InoSV660N)
//     Task_P2Main Inputs/GMotion.arrAxisCtrl[123].Io.DigitalInputs <-> Inputs/Digital inputs
//     Task_P2Main Inputs/GMotion.iActTorque_D[123] <-> Inputs/Torque actual value
//     Task_P2Main Inputs/IO.Network3_OP[18] <-> InfoData/State
//   DPPLC/DPPLC Instance <-> Device 3 (EtherCAT)/Box 2 (CU1128)/Term 44 (CU1128-C)/P2M3尾卷夹电芯旋转（126） (InoSV660N)
//     Task_P2Main Inputs/GMotion.arrAxisCtrl[126].Io.DigitalInputs <-> Inputs/Digital inputs
//     Task_P2Main Inputs/GMotion.iActTorque_D[126] <-> Inputs/Torque actual value
//     Task_P2Main Inputs/IO.Network3_OP[21] <-> InfoData/State
//   DPPLC/DPPLC Instance <-> Device 3 (EtherCAT)/Box 2 (CU1128)/Term 44 (CU1128-C)/P2M3左压刀升降 [120](InoSV660N)
//     Task_P2Main Inputs/GMotion.arrAxisCtrl[120].Io.DigitalInputs <-> Inputs/Digital inputs
//     Task_P2Main Inputs/GMotion.iActTorque_D[120] <-> Inputs/Torque actual value
//     Task_P2Main Inputs/IO.Network3_OP[39] <-> InfoData/State
//   DPPLC/DPPLC Instance <-> Device 3 (EtherCAT)/Box 2 (CU1128)/Term 44 (CU1128-C)/P2M3左压刀开合[119] (InoSV660N)
//     Task_P2Main Inputs/GMotion.arrAxisCtrl[119].Io.DigitalInputs <-> Inputs/Digital inputs
//     Task_P2Main Inputs/GMotion.iActTorque_D[119] <-> Inputs/Torque actual value
//     Task_P2Main Inputs/IO.Network3_OP[38] <-> InfoData/State
//   DPPLC/DPPLC Instance <-> Device 3 (EtherCAT)/Box 2 (CU1128)/Term 44 (CU1128-C)/P2M3拉胶升降[136](InoSV660N)
//     Task_P2Main Inputs/GMotion.arrAxisCtrl[136].Io.DigitalInputs <-> Inputs/Digital inputs
//     Task_P2Main Inputs/GMotion.iActTorque_D[136] <-> Inputs/Torque actual value
//     Task_P2Main Inputs/IO.Network3_OP[33] <-> InfoData/State
//   DPPLC/DPPLC Instance <-> Device 3 (EtherCAT)/Box 2 (CU1128)/Term 44 (CU1128-C)/P2M3正极叠台搬运升降（97）(InoSV660N)
//     Task_P2Main Inputs/GMotion.arrAxisCtrl[97].Io.DigitalInputs <-> Inputs/Digital inputs
//     Task_P2Main Inputs/GMotion.iActTorque_D[97] <-> Inputs/Torque actual value
//     Task_P2Main Inputs/IO.Network3_OP[7] <-> InfoData/State
//   DPPLC/DPPLC Instance <-> Device 3 (EtherCAT)/Box 2 (CU1128)/Term 44 (CU1128-C)/P2M3正极叠台搬运平移1（96） (CDHD)
//     Task_P2Main Inputs/GMotion.arrAxisCtrl[96].Io.DigitalInputs <-> TxPDO 4/Digital inputs
//     Task_P2Main Inputs/GMotion.iActTorque_D[96] <-> TxPDO 1/Torque Actual Value
//     Task_P2Main Inputs/IO.Network3_OP[11] <-> InfoData/State
//   DPPLC/DPPLC Instance <-> Device 3 (EtherCAT)/Box 2 (CU1128)/Term 44 (CU1128-C)/P2M3正极纠偏平台X1（98） (InoSV660N)
//     Task_P2Main Inputs/GMotion.arrAxisCtrl[98].Io.DigitalInputs <-> Inputs/Digital inputs
//     Task_P2Main Inputs/GMotion.iActTorque_D[98] <-> Inputs/Torque actual value
//     Task_P2Main Inputs/IO.Network3_OP[9] <-> InfoData/State
//   DPPLC/DPPLC Instance <-> Device 3 (EtherCAT)/Box 2 (CU1128)/Term 44 (CU1128-C)/P2M3正极纠偏平台X2 （99）(InoSV660N)
//     Task_P2Main Inputs/GMotion.arrAxisCtrl[99].Io.DigitalInputs <-> Inputs/Digital inputs
//     Task_P2Main Inputs/GMotion.iActTorque_D[99] <-> Inputs/Torque actual value
//     Task_P2Main Inputs/IO.Network3_OP[14] <-> InfoData/State
//   DPPLC/DPPLC Instance <-> Device 3 (EtherCAT)/Box 2 (CU1128)/Term 44 (CU1128-C)/P2M3正极纠偏平台Y（100） (InoSV660N)
//     Task_P2Main Inputs/GMotion.arrAxisCtrl[100].Io.DigitalInputs <-> Inputs/Digital inputs
//     Task_P2Main Inputs/GMotion.iActTorque_D[100] <-> Inputs/Torque actual value
//     Task_P2Main Inputs/IO.Network3_OP[15] <-> InfoData/State
//   DPPLC/DPPLC Instance <-> Device 3 (EtherCAT)/Box 2 (CU1128)/Term 44 (CU1128-C)/P2M3正极送料分段皮带3（22模切） (InoSV660N)
//     Task_P2Main Inputs/IO.Network3_OP[1] <-> InfoData/State
//   DPPLC/DPPLC Instance <-> Device 3 (EtherCAT)/Box 2 (CU1128)/Term 44 (CU1128-C)/P2M3正极送片搬运升降（94）(InoSV660N)
//     Task_P2Main Inputs/GMotion.arrAxisCtrl[94].Io.DigitalInputs <-> Inputs/Digital inputs
//     Task_P2Main Inputs/GMotion.iActTorque_D[94] <-> Inputs/Torque actual value
//     Task_P2Main Inputs/IO.Network3_OP[5] <-> InfoData/State
//   DPPLC/DPPLC Instance <-> Device 3 (EtherCAT)/Box 2 (CU1128)/Term 44 (CU1128-C)/P2M3正极送片搬运平移（93） (CDHD)
//     Task_P2Main Inputs/GMotion.arrAxisCtrl[93].Io.DigitalInputs <-> TxPDO 4/Digital inputs
//     Task_P2Main Inputs/GMotion.iActTorque_D[93] <-> TxPDO 1/Torque Actual Value
//     Task_P2Main Inputs/IO.Network3_OP[10] <-> InfoData/State
//   DPPLC/DPPLC Instance <-> Device 3 (EtherCAT)/Box 2 (CU1128)/Term 44 (CU1128-C)/P2M3正极送片搬运旋转 （95）(InoSV660N)
//     Task_P2Main Inputs/GMotion.arrAxisCtrl[95].Io.DigitalInputs <-> Inputs/Digital inputs
//     Task_P2Main Inputs/GMotion.iActTorque_D[95] <-> Inputs/Torque actual value
//     Task_P2Main Inputs/IO.Network3_OP[6] <-> InfoData/State
//   DPPLC/DPPLC Instance <-> Device 3 (EtherCAT)/Box 2 (CU1128)/Term 44 (CU1128-C)/P2M3短卷针平移[130] (CL3C-EC808AC)
//     Task_P2Main Inputs/GMotion.arrAxisCtrl[130].Io.DigitalInputs <-> Transmit PDO 1/Digital Inputs
//     Task_P2Main Inputs/IO.Network3_OP[35] <-> InfoData/State
//   DPPLC/DPPLC Instance <-> Device 3 (EtherCAT)/Box 2 (CU1128)/Term 44 (CU1128-C)/P2M3短卷针旋转[132] (CL3C-EC808AC)
//     Task_P2Main Inputs/GMotion.arrAxisCtrl[132].Io.DigitalInputs <-> Transmit PDO 1/Digital Inputs
//     Task_P2Main Inputs/IO.Network3_OP[46] <-> InfoData/State
//   DPPLC/DPPLC Instance <-> Device 3 (EtherCAT)/Box 2 (CU1128)/Term 44 (CU1128-C)/P2M3负极叠台搬运升降[108](InoSV660N)
//     Task_P2Main Inputs/GMotion.arrAxisCtrl[108].Io.DigitalInputs <-> Inputs/Digital inputs
//     Task_P2Main Inputs/GMotion.iActTorque_D[108] <-> Inputs/Torque actual value
//     Task_P2Main Inputs/IO.Network3_OP[45] <-> InfoData/State
//   DPPLC/DPPLC Instance <-> Device 3 (EtherCAT)/Box 2 (CU1128)/Term 44 (CU1128-C)/P2M3负极叠台搬运平移 [107](CDHD)
//     Task_P2Main Inputs/GMotion.arrAxisCtrl[107].Io.DigitalInputs <-> TxPDO 4/Digital inputs
//     Task_P2Main Inputs/GMotion.iActTorque_D[107] <-> TxPDO 1/Torque Actual Value
//     Task_P2Main Inputs/IO.Network3_OP[29] <-> InfoData/State
//   DPPLC/DPPLC Instance <-> Device 3 (EtherCAT)/Box 2 (CU1128)/Term 44 (CU1128-C)/P2M3负极纠偏平台X1[109](InoSV660N)
//     Task_P2Main Inputs/GMotion.arrAxisCtrl[109].Io.DigitalInputs <-> Inputs/Digital inputs
//     Task_P2Main Inputs/GMotion.iActTorque_D[109] <-> Inputs/Torque actual value
//     Task_P2Main Inputs/IO.Network3_OP[30] <-> InfoData/State
//   DPPLC/DPPLC Instance <-> Device 3 (EtherCAT)/Box 2 (CU1128)/Term 44 (CU1128-C)/P2M3负极纠偏平台X2 [110](InoSV660N)
//     Task_P2Main Inputs/GMotion.arrAxisCtrl[110].Io.DigitalInputs <-> Inputs/Digital inputs
//     Task_P2Main Inputs/GMotion.iActTorque_D[110] <-> Inputs/Torque actual value
//     Task_P2Main Inputs/IO.Network3_OP[31] <-> InfoData/State
//   DPPLC/DPPLC Instance <-> Device 3 (EtherCAT)/Box 2 (CU1128)/Term 44 (CU1128-C)/P2M3负极纠偏平台Y[111](InoSV660N)
//     Task_P2Main Inputs/GMotion.arrAxisCtrl[111].Io.DigitalInputs <-> Inputs/Digital inputs
//     Task_P2Main Inputs/GMotion.iActTorque_D[111] <-> Inputs/Torque actual value
//     Task_P2Main Inputs/IO.Network3_OP[32] <-> InfoData/State
//   DPPLC/DPPLC Instance <-> Device 3 (EtherCAT)/Box 2 (CU1128)/Term 44 (CU1128-C)/P2M3负极送料分段皮带3（46模切） (InoSV660N)
//     Task_P2Main Inputs/IO.Network3_OP[16] <-> InfoData/State
//   DPPLC/DPPLC Instance <-> Device 3 (EtherCAT)/Box 2 (CU1128)/Term 44 (CU1128-C)/P2M3负极送片搬运1升降[102](InoSV660N)
//     Task_P2Main Inputs/GMotion.arrAxisCtrl[102].Io.DigitalInputs <-> Inputs/Digital inputs
//     Task_P2Main Inputs/GMotion.iActTorque_D[102] <-> Inputs/Torque actual value
//     Task_P2Main Inputs/IO.Network3_OP[42] <-> InfoData/State
//   DPPLC/DPPLC Instance <-> Device 3 (EtherCAT)/Box 2 (CU1128)/Term 44 (CU1128-C)/P2M3负极送片搬运1平移[101] (CDHD)
//     Task_P2Main Inputs/GMotion.arrAxisCtrl[101].Io.DigitalInputs <-> TxPDO 4/Digital inputs
//     Task_P2Main Inputs/GMotion.iActTorque_D[101] <-> TxPDO 1/Torque Actual Value
//     Task_P2Main Inputs/IO.Network3_OP[27] <-> InfoData/State
//   DPPLC/DPPLC Instance <-> Device 3 (EtherCAT)/Box 2 (CU1128)/Term 44 (CU1128-C)/P2M3负极送片搬运1旋转[103] (InoSV660N)
//     Task_P2Main Inputs/GMotion.arrAxisCtrl[103].Io.DigitalInputs <-> Inputs/Digital inputs
//     Task_P2Main Inputs/GMotion.iActTorque_D[103] <-> Inputs/Torque actual value
//     Task_P2Main Inputs/IO.Network3_OP[43] <-> InfoData/State
//   DPPLC/DPPLC Instance <-> Device 3 (EtherCAT)/Box 2 (CU1128)/Term 44 (CU1128-C)/P2M3负极送片搬运2升降[105](InoSV660N)
//     Task_P2Main Inputs/GMotion.arrAxisCtrl[105].Io.DigitalInputs <-> Inputs/Digital inputs
//     Task_P2Main Inputs/GMotion.iActTorque_D[105] <-> Inputs/Torque actual value
//     Task_P2Main Inputs/IO.Network3_OP[44] <-> InfoData/State
//   DPPLC/DPPLC Instance <-> Device 3 (EtherCAT)/Box 2 (CU1128)/Term 44 (CU1128-C)/P2M3负极送片搬运2平移[104](CDHD)
//     Task_P2Main Inputs/GMotion.arrAxisCtrl[104].Io.DigitalInputs <-> TxPDO 4/Digital inputs
//     Task_P2Main Inputs/GMotion.iActTorque_D[104] <-> TxPDO 1/Torque Actual Value
//     Task_P2Main Inputs/IO.Network3_OP[28] <-> InfoData/State
//   DPPLC/DPPLC Instance <-> Device 3 (EtherCAT)/Box 2 (CU1128)/Term 44 (CU1128-C)/P2M3负极送片皮带（106） (InoSV660N)
//     Task_P2Main Inputs/GMotion.arrAxisCtrl[106].Io.DigitalInputs <-> Inputs/Digital inputs
//     Task_P2Main Inputs/GMotion.iActTorque_D[106] <-> Inputs/Torque actual value
//     Task_P2Main Inputs/IO.Network3_OP[17] <-> InfoData/State
//   DPPLC/DPPLC Instance <-> Device 3 (EtherCAT)/Box 2 (CU1128)/Term 44 (CU1128-C)/P2M3贴胶头进退[135] (InoSV660N)
//     Task_P2Main Inputs/GMotion.arrAxisCtrl[135].Io.DigitalInputs <-> Inputs/Digital inputs
//     Task_P2Main Inputs/GMotion.iActTorque_D[135] <-> Inputs/Torque actual value
//     Task_P2Main Inputs/IO.Network3_OP[26] <-> InfoData/State
//   DPPLC/DPPLC Instance <-> Device 3 (EtherCAT)/Box 2 (CU1128)/Term 44 (CU1128-C)/P2M3长卷针平移 [129](CL3C-EC808AC)
//     Task_P2Main Inputs/GMotion.arrAxisCtrl[129].Io.DigitalInputs <-> Transmit PDO 1/Digital Inputs
//     Task_P2Main Inputs/IO.Network3_OP[34] <-> InfoData/State
//   DPPLC/DPPLC Instance <-> Device 3 (EtherCAT)/Box 2 (CU1128)/Term 44 (CU1128-C)/P2M3长卷针旋转[131](CL3C-EC808AC)
//     Task_P2Main Inputs/GMotion.arrAxisCtrl[131].Io.DigitalInputs <-> Transmit PDO 1/Digital Inputs
//     Task_P2Main Inputs/IO.Network3_OP[36] <-> InfoData/State
//   DPPLC/DPPLC Instance <-> Device 3 (EtherCAT)/Box 2 (CU1128)/Term 44 (CU1128-C)/P2M3隔膜尾部纠偏 （114）(InoSV660N)
//     Task_P2Main Inputs/GMotion.arrAxisCtrl[114].Io.DigitalInputs <-> Inputs/Digital inputs
//     Task_P2Main Inputs/GMotion.iActTorque_D[114] <-> Inputs/Torque actual value
//     Task_P2Main Inputs/IO.Network3_OP[8] <-> InfoData/State
//   DPPLC/DPPLC Instance <-> Device 3 (EtherCAT)/Box 2 (CU1128)/Term 44 (CU1128-C)/P2M3隔膜平移（117） (CDHD)
//     Task_P2Main Inputs/GMotion.arrAxisCtrl[117].Io.DigitalInputs <-> TxPDO 4/Digital inputs
//     Task_P2Main Inputs/GMotion.iActTorque_D[117] <-> TxPDO 1/Torque Actual Value
//     Task_P2Main Inputs/IO.Network3_OP[12] <-> InfoData/State
//   DPPLC/DPPLC Instance <-> Device 3 (EtherCAT)/Box 2 (CU1128)/Term 44 (CU1128-C)/P2M3隔膜摆杆张力（115） (InoSV660N)
//     Task_P2M3 Outputs/GMotion.iTargetTorque[3] <-> Outputs/Target torque
//     Task_P2Main Inputs/GMotion.arrAxisCtrl[115].Io.DigitalInputs <-> Inputs/Digital inputs
//     Task_P2Main Inputs/GMotion.iActTorque_D[115] <-> Inputs/Torque actual value
//     Task_P2Main Inputs/IO.Network3_OP[3] <-> InfoData/State
//     Task_P3 Outputs/GMotion.iMaxProfileVelo[3] <-> Outputs/Max profile velocity
//     Task_P3 Outputs/GMotion.iNegtiveTorqueLimits[3] <-> Outputs/Negative torque limit value
//     Task_P3 Outputs/GMotion.iPostiveTorqueLimits[3] <-> Outputs/Positive torque limit value
//     Task_P3 Outputs/GMotion.iSetDriveMode[3] <-> Outputs/Modes of operation
//   DPPLC/DPPLC Instance <-> Device 3 (EtherCAT)/Box 2 (CU1128)/Term 44 (CU1128-C)/P2M3隔膜放卷纠偏（113）(InoSV660N)
//     Task_P2Main Inputs/GMotion.arrAxisCtrl[113].Io.DigitalInputs <-> Inputs/Digital inputs
//     Task_P2Main Inputs/GMotion.iActTorque_D[113] <-> Inputs/Torque actual value
//     Task_P2Main Inputs/IO.Network3_OP[2] <-> InfoData/State
//   DPPLC/DPPLC Instance <-> Device 3 (EtherCAT)/Box 2 (CU1128)/Term 44 (CU1128-C)/P2M3隔膜放卷（112） (InoSV660N)
//     Task_P2Main Inputs/GMotion.arrAxisCtrl[112].Io.DigitalInputs <-> Inputs/Digital inputs
//     Task_P2Main Inputs/GMotion.iActTorque_D[112] <-> Inputs/Torque actual value
//     Task_P2Main Inputs/IO.Network3_OP[4] <-> InfoData/State
//   DPPLC/DPPLC Instance <-> Device 3 (EtherCAT)/Box 2 (CU1128)/Term 44 (CU1128-C)/P2M3隔膜缓存（116） (CDHD)
//     Task_P2Main Inputs/GMotion.arrAxisCtrl[116].Io.DigitalInputs <-> TxPDO 4/Digital inputs
//     Task_P2Main Inputs/GMotion.iActTorque_D[116] <-> TxPDO 1/Torque Actual Value
//     Task_P2Main Inputs/IO.Network3_OP[13] <-> InfoData/State
//   DPPLC/DPPLC Instance <-> Device 3 (EtherCAT)/Box 2 (CU1128)/一号叠片IO耦合器(GSIO-A-ECC)
//     Task_P2Main Inputs/IO.AI30[{1..4}] <-> AI301/Analog Inputs/Channel {1..4}  (4 links)
//     Task_P2Main Inputs/IO.I301[10] <-> I301/Digital Inputs/Channel 10
//     Task_P2Main Inputs/IO.I301[11] <-> I301/Digital Inputs/Channel 11
//     Task_P2Main Inputs/IO.I301[12] <-> I301/Digital Inputs/Channel 12
//     Task_P2Main Inputs/IO.I301[13] <-> I301/Digital Inputs/Channel 13
//     Task_P2Main Inputs/IO.I301[14] <-> I301/Digital Inputs/Channel 14
//     Task_P2Main Inputs/IO.I301[15] <-> I301/Digital Inputs/Channel 15
//     Task_P2Main Inputs/IO.I301[16] <-> I301/Digital Inputs/Channel 16
//     Task_P2Main Inputs/IO.I301[1] <-> I301/Digital Inputs/Channel 1
//     Task_P2Main Inputs/IO.I301[2] <-> I301/Digital Inputs/Channel 2
//     Task_P2Main Inputs/IO.I301[3] <-> I301/Digital Inputs/Channel 3
//     Task_P2Main Inputs/IO.I301[4] <-> I301/Digital Inputs/Channel 4
//     Task_P2Main Inputs/IO.I301[5] <-> I301/Digital Inputs/Channel 5
//     Task_P2Main Inputs/IO.I301[6] <-> I301/Digital Inputs/Channel 6
//     Task_P2Main Inputs/IO.I301[7] <-> I301/Digital Inputs/Channel 7
//     Task_P2Main Inputs/IO.I301[8] <-> I301/Digital Inputs/Channel 8
//     Task_P2Main Inputs/IO.I301[9] <-> I301/Digital Inputs/Channel 9
//     Task_P2Main Inputs/IO.I302[10] <-> I302/Digital Inputs/Channel 10
//     Task_P2Main Inputs/IO.I302[11] <-> I302/Digital Inputs/Channel 11
//     Task_P2Main Inputs/IO.I302[12] <-> I302/Digital Inputs/Channel 12
//     Task_P2Main Inputs/IO.I302[13] <-> I302/Digital Inputs/Channel 13
//     Task_P2Main Inputs/IO.I302[14] <-> I302/Digital Inputs/Channel 14
//     Task_P2Main Inputs/IO.I302[15] <-> I302/Digital Inputs/Channel 15
//     Task_P2Main Inputs/IO.I302[16] <-> I302/Digital Inputs/Channel 16
//     Task_P2Main Inputs/IO.I302[1] <-> I302/Digital Inputs/Channel 1
//     Task_P2Main Inputs/IO.I302[2] <-> I302/Digital Inputs/Channel 2
//     Task_P2Main Inputs/IO.I302[3] <-> I302/Digital Inputs/Channel 3
//     Task_P2Main Inputs/IO.I302[4] <-> I302/Digital Inputs/Channel 4
//     Task_P2Main Inputs/IO.I302[5] <-> I302/Digital Inputs/Channel 5
//     Task_P2Main Inputs/IO.I302[6] <-> I302/Digital Inputs/Channel 6
//     Task_P2Main Inputs/IO.I302[7] <-> I302/Digital Inputs/Channel 7
//     Task_P2Main Inputs/IO.I302[8] <-> I302/Digital Inputs/Channel 8
//     Task_P2Main Inputs/IO.I302[9] <-> I302/Digital Inputs/Channel 9
//     Task_P2Main Inputs/IO.I303[10] <-> I303/Digital Inputs/Channel 10
//     Task_P2Main Inputs/IO.I303[11] <-> I303/Digital Inputs/Channel 11
//     Task_P2Main Inputs/IO.I303[12] <-> I303/Digital Inputs/Channel 12
//     Task_P2Main Inputs/IO.I303[13] <-> I303/Digital Inputs/Channel 13
//     Task_P2Main Inputs/IO.I303[14] <-> I303/Digital Inputs/Channel 14
//     Task_P2Main Inputs/IO.I303[15] <-> I303/Digital Inputs/Channel 15
//     Task_P2Main Inputs/IO.I303[16] <-> I303/Digital Inputs/Channel 16
//     Task_P2Main Inputs/IO.I303[1] <-> I303/Digital Inputs/Channel 1
//     Task_P2Main Inputs/IO.I303[2] <-> I303/Digital Inputs/Channel 2
//     Task_P2Main Inputs/IO.I303[3] <-> I303/Digital Inputs/Channel 3
//     Task_P2Main Inputs/IO.I303[4] <-> I303/Digital Inputs/Channel 4
//     Task_P2Main Inputs/IO.I303[5] <-> I303/Digital Inputs/Channel 5
//     Task_P2Main Inputs/IO.I303[6] <-> I303/Digital Inputs/Channel 6
//     Task_P2Main Inputs/IO.I303[7] <-> I303/Digital Inputs/Channel 7
//     Task_P2Main Inputs/IO.I303[8] <-> I303/Digital Inputs/Channel 8
//     Task_P2Main Inputs/IO.I303[9] <-> I303/Digital Inputs/Channel 9
//     Task_P2Main Inputs/IO.I304[10] <-> I304/Digital Inputs/Channel 10
//     Task_P2Main Inputs/IO.I304[11] <-> I304/Digital Inputs/Channel 11
//     Task_P2Main Inputs/IO.I304[12] <-> I304/Digital Inputs/Channel 12
//     Task_P2Main Inputs/IO.I304[13] <-> I304/Digital Inputs/Channel 13
//     Task_P2Main Inputs/IO.I304[14] <-> I304/Digital Inputs/Channel 14
//     Task_P2Main Inputs/IO.I304[15] <-> I304/Digital Inputs/Channel 15
//     Task_P2Main Inputs/IO.I304[16] <-> I304/Digital Inputs/Channel 16
//     Task_P2Main Inputs/IO.I304[1] <-> I304/Digital Inputs/Channel 1
//     Task_P2Main Inputs/IO.I304[2] <-> I304/Digital Inputs/Channel 2
//     Task_P2Main Inputs/IO.I304[3] <-> I304/Digital Inputs/Channel 3
//     Task_P2Main Inputs/IO.I304[4] <-> I304/Digital Inputs/Channel 4
//     Task_P2Main Inputs/IO.I304[5] <-> I304/Digital Inputs/Channel 5
//     Task_P2Main Inputs/IO.I304[6] <-> I304/Digital Inputs/Channel 6
//     Task_P2Main Inputs/IO.I304[7] <-> I304/Digital Inputs/Channel 7
//     Task_P2Main Inputs/IO.I304[8] <-> I304/Digital Inputs/Channel 8
//     Task_P2Main Inputs/IO.I304[9] <-> I304/Digital Inputs/Channel 9
//     Task_P2Main Inputs/IO.I305[10] <-> I305/Digital Inputs/Channel 10
//     Task_P2Main Inputs/IO.I305[11] <-> I305/Digital Inputs/Channel 11
//     Task_P2Main Inputs/IO.I305[12] <-> I305/Digital Inputs/Channel 12
//     Task_P2Main Inputs/IO.I305[13] <-> I305/Digital Inputs/Channel 13
//     Task_P2Main Inputs/IO.I305[14] <-> I305/Digital Inputs/Channel 14
//     Task_P2Main Inputs/IO.I305[15] <-> I305/Digital Inputs/Channel 15
//     Task_P2Main Inputs/IO.I305[16] <-> I305/Digital Inputs/Channel 16
//     Task_P2Main Inputs/IO.I305[1] <-> I305/Digital Inputs/Channel 1
//     Task_P2Main Inputs/IO.I305[2] <-> I305/Digital Inputs/Channel 2
//     Task_P2Main Inputs/IO.I305[3] <-> I305/Digital Inputs/Channel 3
//     Task_P2Main Inputs/IO.I305[4] <-> I305/Digital Inputs/Channel 4
//     Task_P2Main Inputs/IO.I305[5] <-> I305/Digital Inputs/Channel 5
//     Task_P2Main Inputs/IO.I305[6] <-> I305/Digital Inputs/Channel 6
//     Task_P2Main Inputs/IO.I305[7] <-> I305/Digital Inputs/Channel 7
//     Task_P2Main Inputs/IO.I305[8] <-> I305/Digital Inputs/Channel 8
//     Task_P2Main Inputs/IO.I305[9] <-> I305/Digital Inputs/Channel 9
//     Task_P2Main Inputs/IO.I306[10] <-> I306/Digital Inputs/Channel 10
//     Task_P2Main Inputs/IO.I306[11] <-> I306/Digital Inputs/Channel 11
//     Task_P2Main Inputs/IO.I306[12] <-> I306/Digital Inputs/Channel 12
//     Task_P2Main Inputs/IO.I306[13] <-> I306/Digital Inputs/Channel 13
//     Task_P2Main Inputs/IO.I306[14] <-> I306/Digital Inputs/Channel 14
//     Task_P2Main Inputs/IO.I306[15] <-> I306/Digital Inputs/Channel 15
//     Task_P2Main Inputs/IO.I306[16] <-> I306/Digital Inputs/Channel 16
//     Task_P2Main Inputs/IO.I306[1] <-> I306/Digital Inputs/Channel 1
//     Task_P2Main Inputs/IO.I306[2] <-> I306/Digital Inputs/Channel 2
//     Task_P2Main Inputs/IO.I306[3] <-> I306/Digital Inputs/Channel 3
//     Task_P2Main Inputs/IO.I306[4] <-> I306/Digital Inputs/Channel 4
//     Task_P2Main Inputs/IO.I306[5] <-> I306/Digital Inputs/Channel 5
//     Task_P2Main Inputs/IO.I306[6] <-> I306/Digital Inputs/Channel 6
//     Task_P2Main Inputs/IO.I306[7] <-> I306/Digital Inputs/Channel 7
//     Task_P2Main Inputs/IO.I306[8] <-> I306/Digital Inputs/Channel 8
//     Task_P2Main Inputs/IO.I306[9] <-> I306/Digital Inputs/Channel 9
//     Task_P2Main Inputs/IO.I307[10] <-> I307/Digital Inputs/Channel 10
//     Task_P2Main Inputs/IO.I307[11] <-> I307/Digital Inputs/Channel 11
//     Task_P2Main Inputs/IO.I307[12] <-> I307/Digital Inputs/Channel 12
//     Task_P2Main Inputs/IO.I307[13] <-> I307/Digital Inputs/Channel 13
//     Task_P2Main Inputs/IO.I307[14] <-> I307/Digital Inputs/Channel 14
//     Task_P2Main Inputs/IO.I307[15] <-> I307/Digital Inputs/Channel 15
//     Task_P2Main Inputs/IO.I307[16] <-> I307/Digital Inputs/Channel 16
//     Task_P2Main Inputs/IO.I307[1] <-> I307/Digital Inputs/Channel 1
//     Task_P2Main Inputs/IO.I307[2] <-> I307/Digital Inputs/Channel 2
//     Task_P2Main Inputs/IO.I307[3] <-> I307/Digital Inputs/Channel 3
//     Task_P2Main Inputs/IO.I307[4] <-> I307/Digital Inputs/Channel 4
//     Task_P2Main Inputs/IO.I307[5] <-> I307/Digital Inputs/Channel 5
//     Task_P2Main Inputs/IO.I307[6] <-> I307/Digital Inputs/Channel 6
//     Task_P2Main Inputs/IO.I307[7] <-> I307/Digital Inputs/Channel 7
//     Task_P2Main Inputs/IO.I307[8] <-> I307/Digital Inputs/Channel 8
//     Task_P2Main Inputs/IO.I307[9] <-> I307/Digital Inputs/Channel 9
//     Task_P2Main Inputs/IO.I308[10] <-> I308/Digital Inputs/Channel 10
//     Task_P2Main Inputs/IO.I308[11] <-> I308/Digital Inputs/Channel 11
//     Task_P2Main Inputs/IO.I308[12] <-> I308/Digital Inputs/Channel 12
//     Task_P2Main Inputs/IO.I308[13] <-> I308/Digital Inputs/Channel 13
//     Task_P2Main Inputs/IO.I308[14] <-> I308/Digital Inputs/Channel 14
//     Task_P2Main Inputs/IO.I308[15] <-> I308/Digital Inputs/Channel 15
//     Task_P2Main Inputs/IO.I308[16] <-> I308/Digital Inputs/Channel 16
//     Task_P2Main Inputs/IO.I308[1] <-> I308/Digital Inputs/Channel 1
//     Task_P2Main Inputs/IO.I308[2] <-> I308/Digital Inputs/Channel 2
//     Task_P2Main Inputs/IO.I308[3] <-> I308/Digital Inputs/Channel 3
//     Task_P2Main Inputs/IO.I308[4] <-> I308/Digital Inputs/Channel 4
//     Task_P2Main Inputs/IO.I308[5] <-> I308/Digital Inputs/Channel 5
//     Task_P2Main Inputs/IO.I308[6] <-> I308/Digital Inputs/Channel 6
//     Task_P2Main Inputs/IO.I308[7] <-> I308/Digital Inputs/Channel 7
//     Task_P2Main Inputs/IO.I308[8] <-> I308/Digital Inputs/Channel 8
//     Task_P2Main Inputs/IO.I308[9] <-> I308/Digital Inputs/Channel 9
//     Task_P2Main Inputs/IO.I309[10] <-> I309/Digital Inputs/Channel 10
//     Task_P2Main Inputs/IO.I309[11] <-> I309/Digital Inputs/Channel 11
//     Task_P2Main Inputs/IO.I309[12] <-> I309/Digital Inputs/Channel 12
//     Task_P2Main Inputs/IO.I309[13] <-> I309/Digital Inputs/Channel 13
//     Task_P2Main Inputs/IO.I309[14] <-> I309/Digital Inputs/Channel 14
//     Task_P2Main Inputs/IO.I309[15] <-> I309/Digital Inputs/Channel 15
//     Task_P2Main Inputs/IO.I309[16] <-> I309/Digital Inputs/Channel 16
//     Task_P2Main Inputs/IO.I309[1] <-> I309/Digital Inputs/Channel 1
//     Task_P2Main Inputs/IO.I309[2] <-> I309/Digital Inputs/Channel 2
//     Task_P2Main Inputs/IO.I309[3] <-> I309/Digital Inputs/Channel 3
//     Task_P2Main Inputs/IO.I309[4] <-> I309/Digital Inputs/Channel 4
//     Task_P2Main Inputs/IO.I309[5] <-> I309/Digital Inputs/Channel 5
//     Task_P2Main Inputs/IO.I309[6] <-> I309/Digital Inputs/Channel 6
//     Task_P2Main Inputs/IO.I309[7] <-> I309/Digital Inputs/Channel 7
//     Task_P2Main Inputs/IO.I309[8] <-> I309/Digital Inputs/Channel 8
//     Task_P2Main Inputs/IO.I309[9] <-> I309/Digital Inputs/Channel 9
//     Task_P2Main Inputs/IO.Network4_OP[3] <-> InfoData/State
//     Task_P2Main Outputs/IO.Q301[10] <-> Q301/Digital Outputs/Channel 10
//     Task_P2Main Outputs/IO.Q301[11] <-> Q301/Digital Outputs/Channel 11
//     Task_P2Main Outputs/IO.Q301[12] <-> Q301/Digital Outputs/Channel 12
//     Task_P2Main Outputs/IO.Q301[13] <-> Q301/Digital Outputs/Channel 13
//     Task_P2Main Outputs/IO.Q301[14] <-> Q301/Digital Outputs/Channel 14
//     Task_P2Main Outputs/IO.Q301[15] <-> Q301/Digital Outputs/Channel 15
//     Task_P2Main Outputs/IO.Q301[16] <-> Q301/Digital Outputs/Channel 16
//     Task_P2Main Outputs/IO.Q301[1] <-> Q301/Digital Outputs/Channel 1
//     Task_P2Main Outputs/IO.Q301[2] <-> Q301/Digital Outputs/Channel 2
//     Task_P2Main Outputs/IO.Q301[5] <-> Q301/Digital Outputs/Channel 5
//     Task_P2Main Outputs/IO.Q301[6] <-> Q301/Digital Outputs/Channel 6
//     Task_P2Main Outputs/IO.Q301[7] <-> Q301/Digital Outputs/Channel 7
//     Task_P2Main Outputs/IO.Q301[8] <-> Q301/Digital Outputs/Channel 8
//     Task_P2Main Outputs/IO.Q301[9] <-> Q301/Digital Outputs/Channel 9
//     Task_P2Main Outputs/IO.Q302[10] <-> Q302/Digital Outputs/Channel 10
//     Task_P2Main Outputs/IO.Q302[11] <-> Q302/Digital Outputs/Channel 11
//     Task_P2Main Outputs/IO.Q302[12] <-> Q302/Digital Outputs/Channel 12
//     Task_P2Main Outputs/IO.Q302[13] <-> Q302/Digital Outputs/Channel 13
//     Task_P2Main Outputs/IO.Q302[14] <-> Q302/Digital Outputs/Channel 14
//     Task_P2Main Outputs/IO.Q302[15] <-> Q302/Digital Outputs/Channel 15
//     Task_P2Main Outputs/IO.Q302[16] <-> Q302/Digital Outputs/Channel 16
//     Task_P2Main Outputs/IO.Q302[3] <-> Q302/Digital Outputs/Channel 3
//     Task_P2Main Outputs/IO.Q302[4] <-> Q302/Digital Outputs/Channel 4
//     Task_P2Main Outputs/IO.Q302[5] <-> Q302/Digital Outputs/Channel 5
//     Task_P2Main Outputs/IO.Q302[6] <-> Q302/Digital Outputs/Channel 6
//     Task_P2Main Outputs/IO.Q302[7] <-> Q302/Digital Outputs/Channel 7
//     Task_P2Main Outputs/IO.Q302[8] <-> Q302/Digital Outputs/Channel 8
//     Task_P2Main Outputs/IO.Q302[9] <-> Q302/Digital Outputs/Channel 9
//     Task_P2Main Outputs/IO.Q303[10] <-> Q303/Digital Outputs/Channel 10
//     Task_P2Main Outputs/IO.Q303[11] <-> Q303/Digital Outputs/Channel 11
//     Task_P2Main Outputs/IO.Q303[12] <-> Q303/Digital Outputs/Channel 12
//     Task_P2Main Outputs/IO.Q303[13] <-> Q303/Digital Outputs/Channel 13
//     Task_P2Main Outputs/IO.Q303[14] <-> Q303/Digital Outputs/Channel 14
//     Task_P2Main Outputs/IO.Q303[15] <-> Q303/Digital Outputs/Channel 15
//     Task_P2Main Outputs/IO.Q303[16] <-> Q303/Digital Outputs/Channel 16
//     Task_P2Main Outputs/IO.Q303[1] <-> Q303/Digital Outputs/Channel 1
//     Task_P2Main Outputs/IO.Q303[2] <-> Q303/Digital Outputs/Channel 2
//     Task_P2Main Outputs/IO.Q303[3] <-> Q303/Digital Outputs/Channel 3
//     Task_P2Main Outputs/IO.Q303[4] <-> Q303/Digital Outputs/Channel 4
//     Task_P2Main Outputs/IO.Q303[5] <-> Q303/Digital Outputs/Channel 5
//     Task_P2Main Outputs/IO.Q303[6] <-> Q303/Digital Outputs/Channel 6
//     Task_P2Main Outputs/IO.Q303[7] <-> Q303/Digital Outputs/Channel 7
//     Task_P2Main Outputs/IO.Q303[8] <-> Q303/Digital Outputs/Channel 8
//     Task_P2Main Outputs/IO.Q303[9] <-> Q303/Digital Outputs/Channel 9
//     Task_P2Main Outputs/IO.Q304[10] <-> Q304/Digital Outputs/Channel 10
//     Task_P2Main Outputs/IO.Q304[11] <-> Q304/Digital Outputs/Channel 11
//     Task_P2Main Outputs/IO.Q304[12] <-> Q304/Digital Outputs/Channel 12
//     Task_P2Main Outputs/IO.Q304[13] <-> Q304/Digital Outputs/Channel 13
//     Task_P2Main Outputs/IO.Q304[14] <-> Q304/Digital Outputs/Channel 14
//     Task_P2Main Outputs/IO.Q304[15] <-> Q304/Digital Outputs/Channel 15
//     Task_P2Main Outputs/IO.Q304[16] <-> Q304/Digital Outputs/Channel 16
//     Task_P2Main Outputs/IO.Q304[1] <-> Q304/Digital Outputs/Channel 1
//     Task_P2Main Outputs/IO.Q304[2] <-> Q304/Digital Outputs/Channel 2
//     Task_P2Main Outputs/IO.Q304[3] <-> Q304/Digital Outputs/Channel 3
//     Task_P2Main Outputs/IO.Q304[4] <-> Q304/Digital Outputs/Channel 4
//     Task_P2Main Outputs/IO.Q304[5] <-> Q304/Digital Outputs/Channel 5
//     Task_P2Main Outputs/IO.Q304[6] <-> Q304/Digital Outputs/Channel 6
//     Task_P2Main Outputs/IO.Q304[7] <-> Q304/Digital Outputs/Channel 7
//     Task_P2Main Outputs/IO.Q304[8] <-> Q304/Digital Outputs/Channel 8
//     Task_P2Main Outputs/IO.Q304[9] <-> Q304/Digital Outputs/Channel 9
//     Task_P2Main Outputs/IO.Q305[10] <-> Q305/Digital Outputs/Channel 10
//     Task_P2Main Outputs/IO.Q305[11] <-> Q305/Digital Outputs/Channel 11
//     Task_P2Main Outputs/IO.Q305[12] <-> Q305/Digital Outputs/Channel 12
//     Task_P2Main Outputs/IO.Q305[13] <-> Q305/Digital Outputs/Channel 13
//     Task_P2Main Outputs/IO.Q305[14] <-> Q305/Digital Outputs/Channel 14
//     Task_P2Main Outputs/IO.Q305[15] <-> Q305/Digital Outputs/Channel 15
//     Task_P2Main Outputs/IO.Q305[16] <-> Q305/Digital Outputs/Channel 16
//     Task_P2Main Outputs/IO.Q305[1] <-> Q305/Digital Outputs/Channel 1
//     Task_P2Main Outputs/IO.Q305[2] <-> Q305/Digital Outputs/Channel 2
//     Task_P2Main Outputs/IO.Q305[3] <-> Q305/Digital Outputs/Channel 3
//     Task_P2Main Outputs/IO.Q305[4] <-> Q305/Digital Outputs/Channel 4
//     Task_P2Main Outputs/IO.Q305[5] <-> Q305/Digital Outputs/Channel 5
//     Task_P2Main Outputs/IO.Q305[6] <-> Q305/Digital Outputs/Channel 6
//     Task_P2Main Outputs/IO.Q305[7] <-> Q305/Digital Outputs/Channel 7
//     Task_P2Main Outputs/IO.Q305[8] <-> Q305/Digital Outputs/Channel 8
//     Task_P2Main Outputs/IO.Q305[9] <-> Q305/Digital Outputs/Channel 9
//     Task_P2Main Outputs/IO.Q306[10] <-> Q306/Digital Outputs/Channel 10
//     Task_P2Main Outputs/IO.Q306[11] <-> Q306/Digital Outputs/Channel 11
//     Task_P2Main Outputs/IO.Q306[12] <-> Q306/Digital Outputs/Channel 12
//     Task_P2Main Outputs/IO.Q306[13] <-> Q306/Digital Outputs/Channel 13
//     Task_P2Main Outputs/IO.Q306[14] <-> Q306/Digital Outputs/Channel 14
//     Task_P2Main Outputs/IO.Q306[15] <-> Q306/Digital Outputs/Channel 15
//     Task_P2Main Outputs/IO.Q306[16] <-> Q306/Digital Outputs/Channel 16
//     Task_P2Main Outputs/IO.Q306[1] <-> Q306/Digital Outputs/Channel 1
//     Task_P2Main Outputs/IO.Q306[2] <-> Q306/Digital Outputs/Channel 2
//     Task_P2Main Outputs/IO.Q306[3] <-> Q306/Digital Outputs/Channel 3
//     Task_P2Main Outputs/IO.Q306[4] <-> Q306/Digital Outputs/Channel 4
//     Task_P2Main Outputs/IO.Q306[5] <-> Q306/Digital Outputs/Channel 5
//     Task_P2Main Outputs/IO.Q306[6] <-> Q306/Digital Outputs/Channel 6
//     Task_P2Main Outputs/IO.Q306[7] <-> Q306/Digital Outputs/Channel 7
//     Task_P2Main Outputs/IO.Q306[8] <-> Q306/Digital Outputs/Channel 8
//     Task_P2Main Outputs/IO.Q306[9] <-> Q306/Digital Outputs/Channel 9
//     Task_P2Main Outputs/IO.Q307[10] <-> Q307/Digital Outputs/Channel 10
//     Task_P2Main Outputs/IO.Q307[11] <-> Q307/Digital Outputs/Channel 11
//     Task_P2Main Outputs/IO.Q307[12] <-> Q307/Digital Outputs/Channel 12
//     Task_P2Main Outputs/IO.Q307[13] <-> Q307/Digital Outputs/Channel 13
//     Task_P2Main Outputs/IO.Q307[14] <-> Q307/Digital Outputs/Channel 14
//     Task_P2Main Outputs/IO.Q307[15] <-> Q307/Digital Outputs/Channel 15
//     Task_P2Main Outputs/IO.Q307[16] <-> Q307/Digital Outputs/Channel 16
//     Task_P2Main Outputs/IO.Q307[1] <-> Q307/Digital Outputs/Channel 1
//     Task_P2Main Outputs/IO.Q307[2] <-> Q307/Digital Outputs/Channel 2
//     Task_P2Main Outputs/IO.Q307[3] <-> Q307/Digital Outputs/Channel 3
//     Task_P2Main Outputs/IO.Q307[4] <-> Q307/Digital Outputs/Channel 4
//     Task_P2Main Outputs/IO.Q307[5] <-> Q307/Digital Outputs/Channel 5
//     Task_P2Main Outputs/IO.Q307[6] <-> Q307/Digital Outputs/Channel 6
//     Task_P2Main Outputs/IO.Q307[7] <-> Q307/Digital Outputs/Channel 7
//     Task_P2Main Outputs/IO.Q307[8] <-> Q307/Digital Outputs/Channel 8
//     Task_P2Main Outputs/IO.Q307[9] <-> Q307/Digital Outputs/Channel 9
//     Task_P2Main Outputs/IO.Q309[10] <-> Q309/Digital Outputs/Channel 10
//     Task_P2Main Outputs/IO.Q309[11] <-> Q309/Digital Outputs/Channel 11
//     Task_P2Main Outputs/IO.Q309[12] <-> Q309/Digital Outputs/Channel 12
//     Task_P2Main Outputs/IO.Q309[13] <-> Q309/Digital Outputs/Channel 13
//     Task_P2Main Outputs/IO.Q309[14] <-> Q309/Digital Outputs/Channel 14
//     Task_P2Main Outputs/IO.Q309[15] <-> Q309/Digital Outputs/Channel 15
//     Task_P2Main Outputs/IO.Q309[16] <-> Q309/Digital Outputs/Channel 16
//     Task_P2Main Outputs/IO.Q309[1] <-> Q309/Digital Outputs/Channel 1
//     Task_P2Main Outputs/IO.Q309[2] <-> Q309/Digital Outputs/Channel 2
//     Task_P2Main Outputs/IO.Q309[3] <-> Q309/Digital Outputs/Channel 3
//     Task_P2Main Outputs/IO.Q309[4] <-> Q309/Digital Outputs/Channel 4
//     Task_P2Main Outputs/IO.Q309[5] <-> Q309/Digital Outputs/Channel 5
//     Task_P2Main Outputs/IO.Q309[6] <-> Q309/Digital Outputs/Channel 6
//     Task_P2Main Outputs/IO.Q309[7] <-> Q309/Digital Outputs/Channel 7
//     Task_P2Main Outputs/IO.Q309[8] <-> Q309/Digital Outputs/Channel 8
//     Task_P2Main Outputs/IO.Q309[9] <-> Q309/Digital Outputs/Channel 9
//     Task_P3 Outputs/IO.Q308[{1..16}] <-> Q308/Digital Outputs/Channel {1..16}  (16 links)
//   DPPLC/DPPLC Instance <-> Device 3 (EtherCAT)/Box 2 (CU1128)/一号烤箱温控器1(SM693H-1*H)
//     Task_P2Main Inputs/IO.Network4_OP[7] <-> InfoData/State
//     Task_P3 Inputs/P3Temperature.TempPVs[10]/iPV1 <-> Module 4 (RTD.8CH)/RTD.8Ch/Channel2
//     Task_P3 Inputs/P3Temperature.TempPVs[11]/iPV1 <-> Module 4 (RTD.8CH)/RTD.8Ch/Channel3
//     Task_P3 Inputs/P3Temperature.TempPVs[12]/iPV1 <-> Module 4 (RTD.8CH)/RTD.8Ch/Channel4
//     Task_P3 Inputs/P3Temperature.TempPVs[13]/iPV1 <-> Module 4 (RTD.8CH)/RTD.8Ch/Channel5
//     Task_P3 Inputs/P3Temperature.TempPVs[14]/iPV1 <-> Module 4 (RTD.8CH)/RTD.8Ch/Channel6
//     Task_P3 Inputs/P3Temperature.TempPVs[15]/iPV1 <-> Module 4 (RTD.8CH)/RTD.8Ch/Channel7
//     Task_P3 Inputs/P3Temperature.TempPVs[16]/iPV1 <-> Module 4 (RTD.8CH)/RTD.8Ch/Channel8
//     Task_P3 Inputs/P3Temperature.TempPVs[1]/iPV1 <-> Module 3 (RTD.8CH)/RTD.8Ch/Channel1
//     Task_P3 Inputs/P3Temperature.TempPVs[2]/iPV1 <-> Module 3 (RTD.8CH)/RTD.8Ch/Channel2
//     Task_P3 Inputs/P3Temperature.TempPVs[3]/iPV1 <-> Module 3 (RTD.8CH)/RTD.8Ch/Channel3
//     Task_P3 Inputs/P3Temperature.TempPVs[4]/iPV1 <-> Module 3 (RTD.8CH)/RTD.8Ch/Channel4
